CT_DisAction_2[1](xCycleStartMark:=Cy_lifter.xHP_Valve ,xCycleEndMark:= Cy_lifter.xHP_Delay,xCycleRun:=TRUE, RCycleTime=>ct_show.S01_CY_Lifter_HP);
CT_DisAction_2[2](xCycleStartMark:=Cy_lifter.xWP_Valve ,xCycleEndMark:= Cy_lifter.xWP_Delay,xCycleRun:=TRUE, RCycleTime=>ct_show.S01_CY_Lifter_WP);
CT_DisAction_2[3](xCycleStartMark:=Cy_rotate.xHP_Valve ,xCycleEndMark:= Cy_rotate.xHP_Delay,xCycleRun:=TRUE, RCycleTime=>ct_show.S01_CY_Rotate_HP);
CT_DisAction_2[4](xCycleStartMark:=Cy_rotate.xWP_Valve ,xCycleEndMark:= Cy_rotate.xWP_Delay,xCycleRun:=TRUE, RCycleTime=>ct_show.S01_CY_Rotate_WP);
CT_DisAction_2[5](xCycleStartMark:=Cy_takeClamp1.xHP_Valve ,xCycleEndMark:= Cy_takeClamp1.xHP_Delay,xCycleRun:=TRUE, RCycleTime=>ct_show.S01_Cy_takeClamp12_HP);
CT_DisAction_2[6](xCycleStartMark:=Cy_takeClamp1.xWP_Valve ,xCycleEndMark:= Cy_takeClamp1.xWP_Delay,xCycleRun:=TRUE, RCycleTime=>ct_show.S01_Cy_takeClamp12_WP);
CT_DisAction_2[7](xCycleStartMark:=Cy_takeClamp3.xHP_Valve ,xCycleEndMark:= Cy_takeClamp3.xHP_Delay,xCycleRun:=TRUE, RCycleTime=>ct_show.S01_Cy_takeClamp34_HP);
CT_DisAction_2[8](xCycleStartMark:=Cy_takeClamp3.xWP_Valve ,xCycleEndMark:= Cy_takeClamp3.xWP_Delay,xCycleRun:=TRUE, RCycleTime=>ct_show.S01_Cy_takeClamp34_WP);



//---------------------------------CV运行---------------------------------
 IF Machine_IO.xAutoMode THEN //自动模式下
	 IF station.xRunning THEN
		  Motion_ADD_cv_run[1]:=TRUE;//传送带运行置位
      Motion_ADD_cv_run[2]:=TRUE;   
   END_IF
END_IF
ft_cv(CLK:=station.xRunning AND  Machine_IO.xAutoMode , Q=> );
IF ft_cv.Q THEN
	 Motion_ADD_cv_run[1]:=FALSE;//传送带运行复位
   Motion_ADD_cv_run[2]:=FALSE;  
 END_IF
 
 //--------------------------------数据处理------------------------------
  rt_Clamp1HP(CLK:=Cy_takeClamp1.xHP_Delay, Q=> );
  rt_Clamp2HP(CLK:=Cy_takeClamp3.xHP_Delay , Q=> );
 //IF (rt_Clamp1HP.Q AND  Cy_rotate.xWP_Sensor) OR (rt_Clamp2HP.Q AND Cy_rotate.xHP_Sensor) THEN 	     
 IF station.xRunning AND NOT S05_CircleLine.Axis_Cycleline.xbusy THEN
   IF	 Sensor_Cycleline_on[1] OR (fbmachine[1].xTryRun) THEN
		 CardState[1].A:=TRUE;
		 CardState[1].Card_OK:=TRUE;	
   END_IF
   IF	 Sensor_Cycleline_on[2] OR (fbmachine[1].xTryRun) THEN
	 	 CardState[1].B:=TRUE;
		 CardState[1].Card_OK:=TRUE;	
	 END_IF
END_IF
END_ACTION

ACTION ILC:

//---------------------------------------------------工站可执行-------------------------------------------------------
station.xCanRun := TRUE ;

//---------------------------------------------------气缸动作条件-------------------------------------------
Cy_rotate.xOnILC:=Cy_lifter.xHP_Sensor OR Cy_rotate.xWP_Valve;
Cy_rotate.xOffILC:=Cy_lifter.xHP_Sensor OR Cy_rotate.xHP_Valve;

Cy_takeClamp1.xOnILC:=
Cy_takeClamp1.xOffILC:=TRUE;
                       //Cy_lifter.xWP_Delay 

//Cy_takeClamp2.xOnILC:=
//Cy_takeClamp2.xOffILC:=TRUE;

Cy_takeClamp3.xOnILC:=
Cy_takeClamp3.xOffILC:=TRUE;


//Cy_takeClamp4.xOnILC:=
//Cy_takeClamp4.xOffILC:=TRUE;

Cy_lifter.xOnILC:=NOT S05_CircleLine.Axis_Cycleline.xbusy AND Cy_rotate_on;
Cy_lifter.xOffILC:= TRUE ;
END_ACTION

ACTION TipAuto:

//------------------------------------------------AutoTip General---------------------------------


//------------------------------------------------AutoTip Cylinder--------------------------------

station.adwAutoTip[1].00:=FALSE;	//
station.adwAutoTip[1].01:=FALSE;	//
station.adwAutoTip[1].02:=Cy_rotate.xAutoTip;	       //Cy_rotate 气缸自动中有手动
station.adwAutoTip[1].03:=Cy_takeClamp1.xAutoTip;	   //Cy_takeClamp1 气缸自动中有手动
//station.adwAutoTip[1].04:=Cy_takeClamp2.xAutoTip;	   //Cy_takeClamp2 气缸自动中有手动
station.adwAutoTip[1].05:=Cy_takeClamp3.xAutoTip;	   //Cy_takeClamp3 气缸自动中有手动
//station.adwAutoTip[1].06:=Cy_takeClamp4.xAutoTip;	   //Cy_takeClamp4 气缸自动中有手动
station.adwAutoTip[1].07:=Cy_lifter	.xAutoTip;	     //Cy_lifter 气缸自动中有手动
END_ACTION

ACTION TipManual:
//--------------------------------------------ManualTip------------------------------------------------------
station.adwManualTip[1].00			:=FALSE;//提示1
//-------------------------------------------气缸提示---------------------------------------------------------




/////////////////////////////////////////////////////////////////////////////////////////////////////////////////
END_ACTION

END_PROGRAM

// Device/Application/POUS/02_STATION/S05_CircleLine
PROGRAM S05_CircleLine
VAR_INPUT

		//工站
	station					    : REFERENCE TO FB_Station:=fbStation[5];//工站状态
	cycleTime						: REFERENCE TO FB_CycleTime:= fbStCycleTime[5];	//工站CT
	//伺服
	Axis_Cycleline	    : REFERENCE TO FB_Axis:=fbAxis[1];
END_VAR
VAR
			arTon                 :ARRAY[1..10] OF ton ; 
			arTon_alarm           :ARRAY[1..10] OF ton ; 
		  cycle_data_switch     :R_TRIG;//数据切换信号
		  rt_Ctmark             :R_TRIG;
			i                     :INT;
			Transplant_Can        :BOOL;
			Bowlfeeder_Can        :BOOL;
			Pushcard_Can          :BOOL;
			Takebag_Can           :BOOL;
			Openbag_Can           :BOOL;			
			CT_DisAction          : ARRAY[1..10] OF FB_CycleTime;
			CT_DisAction_1        : ARRAY[1..10] OF FB_CycleTime_1;			
	  	CT_DisAction_2        : ARRAY[1..10] OF FB_CycleTime_2;			
END_VAR

Alarm();
Delay();
FlowAuto();
FlowInit();
General();
ILC();
TipAuto();
TipManual();

ACTION Alarm:
station.adwAlarm[1].00:=station.xInitTimeout;	             //工站初始化超时报警
station.adwAlarm[1].19:=	Axis_Cycleline.xError ;            //轴报错
station.adwAlarm[1].20:=	Axis_Cycleline.xNotPowerOn;         //未使能
station.adwAlarm[1].21:=	Axis_Cycleline.xMoveTimeout;        //定位超时
END_ACTION

ACTION Delay:

//----------------------------------------------动作延时-----------------------------------------------

arTon[1](IN:=  , PT:=T#10S , Q=> , ET=> );//排空计时
arTon[2](IN:=NOT CardState[1].Card_OK AND NOT Axis_Cycleline.xbusy AND xCycle_card_on , PT:=T#10S , Q=> , ET=> );//
arTon[3](IN:=   , PT:=T#60S , Q=> , ET=> );//
//----------------------------------------------报警延时-----------------------------------------------
arTon_alarm[1](IN:=NOT Axis_Cycleline.xbusy  , PT:=T#1S , Q=> , ET=> );//
arTon_alarm[2](IN:= , PT:=T#7S , Q=> , ET=> );//
arTon_alarm[3](IN:= , PT:=T#7S , Q=> , ET=> );//
arTon_alarm[4](IN:= , PT:=T#7S , Q=> , ET=> );//
arTon_alarm[5](IN:=   , PT:=T#60S , Q=> , ET=> );//
arTon_alarm[6](IN:=   , PT:=T#60S , Q=> , ET=> );//

arTon_alarm[7](IN:=   , PT:=T#10S , Q=> , ET=> );//
arTon_alarm[8](IN:=   , PT:=T#60S , Q=> , ET=> );//
arTon_alarm[9](IN:=   , PT:=T#60S , Q=> , ET=> );//
END_ACTION

ACTION FlowAuto:

//-----------------------------------------初始化是否完成判断----------------------------------------------
IF NOT station.xInitDone 
THEN
 	station.iStepAuto:=0;
 	station.xDone:=FALSE;
ELSIF station.xRunning  
THEN
//-----------------------------------------动作步骤--------------------------------------------------------
CASE station.iStepAuto OF	  
	0: //----Home Step，等待启动----
		
		IF station.xDisabled AND station.xCanRun 	AND NOT fbMachine[1].xStopped AND NOT station.xSingleRunning 
		THEN
			station.xDone:=TRUE;//工站完成信号判断
		END_IF
		
	  IF  station.xSingleRunning OR station.xCanRun	AND NOT station.xDone AND NOT station.xDisabled	AND NOT fbMachine[1].xStopped
		THEN
			station.xCycleEnable:=TRUE;
			station.xDone:= FALSE;  
			station.iStepAuto:= 60;
		END_IF

		40://启动前判断运行条件
		IF Axis_Cycleline.xRunILC AND S03_takebag.Axis_Cycleline.xRunILC THEN
	 //  S05_CycleLineMoveCount:= S05_CycleLineMoveCount +1;
	  	station.iStepAuto:= 50;
		END_IF	 
		50://启动
(*		 stData.Axis[1].rMovePosition[2] := stData.Axis[1].rMovePosition[1] +S05_CycleLineMoveCount* gc_rCycleLineSpacing;//200为两个节距
	   Axis_Cycleline.xMoveAuto[2]:=TRUE;//供袋环形线移动
    IF  Axis_Cycleline.xMoveInPos[2] THEN
				station.iStepAuto:= 999;  
		END_IF		
*)
    60:
		IF (Transplant_Can OR S01_transplant.station.xDisabled)
      AND (Bowlfeeder_Can OR S02_bowlFeeder.station.xDisabled) 
      AND (Pushcard_Can OR S04_PushCard.station.xDisabled)
      AND (Takebag_Can OR S03_takebag.station.xDisabled)
      AND (Openbag_Can OR  S06_OpenBag.station.xDisabled) AND NOT Axis_Cycleline.xbusy THEN		
		
		  station.iStepAuto :=70;
		END_IF

	70://数据处理
	IF NOT Axis_Cycleline.xbusy THEN
		Axis_Cycleline.xRelativeAuto:=TRUE;	
	END_IF
	IF Axis_Cycleline.xbusy THEN
		  FOR K :=8 TO 1 BY -1 DO
			CardState[K+1] := CardState[K] ;	
		  END_FOR  
			CardState[1]:=CardState[5]:=CardState[6];	//word 5 数据复位	
			station.iStepAuto :=80;
	END_IF
	80:	//等待完成	 
	  IF  Axis_Cycleline.xRelativeDone1  THEN
	    station.iStepAuto :=999;
		END_IF
	  999://----Single Run Finish----
		station.iStepAuto :=0;
		//station.xDone:=TRUE;
		station.xSingleRunFlag:=FALSE;
		station.xCycleEnable:=FALSE;	
END_CASE

END_IF
END_ACTION

ACTION FlowInit:
IF NOT station.xIniting THEN
  station.iStepInit:=0;    
ELSE
//--------------------------------------------初始化步序----------------------------------
CASE station.iStepInit OF	
 0://  
  	IF station.xIniting THEN	
  	  station.iStepInit:=10;	
  	END_IF	
10://复位数据
			CardState:= zero_card ;
      station.iStepInit := 20 ;		

20://轴上使能
   	Axis_Cycleline.xPowerInit := TRUE ;
    IF 	Axis_Cycleline.xPowerOn THEN 
    		station.iStepInit:=50;	
		END_IF		
50://轴回原点
    Axis_Cycleline.xHomeAuto := TRUE ;
		IF Axis_Cycleline.xHomeDone THEN
    Axis_Cycleline.xHomeAuto := FALSE ;
    		station.iStepInit:=60;	
		END_IF
60://轴去待机位
    Axis_Cycleline.xMoveAuto[1] := TRUE ;
		IF Axis_Cycleline.xMoveInPos[1] THEN 
    		station.iStepInit:=999;	
		END_IF			
999://初始化完成	
	station.iStepInit:=0;
	station.xInitDone:=TRUE;  
END_CASE
END_IF
END_ACTION

ACTION General:
//工站信息处理

(*IF station.xRunning THEN 
	//word 1有料判断，和传送复位
//传送时，数据交替	 
	 cycle_data_switch(CLK:=Axis_Cycleline.xMoveAuto[2], Q=> );
	 IF cycle_data_switch.Q THEN
		 FOR K :=8 TO 1 BY -1 DO
			CardState[K+1] := CardState[K] ;	
		  END_FOR  
		CardState[5]:=CardState[6];	//word 5 数据复位
	 END_IF 
END_IF
*)
//主轴停止状态
Axis_main_ready:=NOT Axis_Cycleline.xbusy;
//主轴上有料判断
IF CardState[1].Card_OK OR CardState[2].Card_OK OR CardState[3].Card_OK OR CardState[4].Card_OK  THEN
	xCycle_card_on:=TRUE;
	ELSE
	xCycle_card_on:=FALSE;	
END_IF
//周边工站完成信号复位
cycle_data_switch(CLK:=Axis_Cycleline.xbusy, Q=> );
IF cycle_data_switch.Q  THEN
	S01_transplant.station.xDone:=FALSE;
	S02_bowlFeeder.station.xDone:=FALSE;
//  S03_takebag.station.xDone:=FALSE;
	S04_PushCard.station.xDone:=FALSE;
//	S06_OpenBag.station.xDone:=FALSE;
END_IF
//自动排空处理
 //xCard_Empty:=TRUE;
 //点动数据，前进一节手动操作
 stData.Axis[1].rRelativeDistance:=gc_rCycleLineSpacing;
 
//CT
rt_Ctmark(CLK:=Axis_Cycleline.xRelativeAuto, Q=>cycleTime.xCycleMark );   
 
CT_DisAction[1](xCycleMark:=Axis_Cycleline.xbusy,xCycleRun:=TRUE,rCycleTime=>);
CT_DisAction[2](xCycleMark:=NOT Bowlfeeder_Can,xCycleRun:=TRUE,rCycleTime=>);
CT_DisAction[3](xCycleMark:=NOT Takebag_Can,xCycleRun:=TRUE,rCycleTime=>);
CT_DisAction[4](xCycleMark:=NOT Pushcard_Can,xCycleRun:=TRUE,rCycleTime=>);
CT_DisAction[5](xCycleMark:=NOT Openbag_Can,xCycleRun:=TRUE,rCycleTime=>);
CT_DisAction[6](xCycleMark:=Axis_Cycleline.xRelativeAuto,xCycleRun:=TRUE, RCycleTime=>ct_show.S05_Total);

CT_DisAction_1[1](xCycleMark:=Axis_Cycleline.xbusy,xCycleRun:=TRUE, RCycleTime=>ct_show.S05_AXIS_Relative);

//工站运行条件可
//S01
IF (CardState[1].Card_OK OR arTon[2].Q OR S01_transplant.station.xDisabled ) AND  S01_transplant.Cy_lifter.xHP_Delay  THEN
	Transplant_Can:=TRUE;
	ELSE
	Transplant_Can:=FALSE;
END_IF
//S02
IF CardState[2].Desiccant_OK OR NOT CardState[2].Card_OK OR S02_bowlFeeder.station.xDisabled THEN
	Bowlfeeder_Can:=TRUE;
	ELSE
	Bowlfeeder_Can:=FALSE;
END_IF
//S03
IF (BagState[1].Takebag_OK OR NOT CardState[2].Card_OK OR S03_takebag.station.xDisabled) AND S03_takebag.Cy_lifter.xHP_Delay  THEN
	Takebag_Can:=TRUE;
	ELSE
	Takebag_Can:=FALSE;
END_IF
//S04
IF (CardState[4].Pushcard_OK OR NOT CardState[4].Card_OK OR S04_PushCard.station.xDisabled) AND S04_PushCard.Cy_push1.xHP_Delay AND S04_PushCard.Cy_push2.xHP_Delay  THEN
	Pushcard_Can:=TRUE;
	ELSE
	Pushcard_Can:=FALSE;
END_IF
//S06
IF BagState[2].Suck_OK OR NOT CardState[3].Card_OK OR S06_OpenBag.station.xDisabled   THEN
	Openbag_Can:=TRUE;
	ELSE
	Openbag_Can:=FALSE;
END_IF
END_ACTION

ACTION ILC:

//---------------------------------------------------工站可执行-------------------------------------------------------
station.xCanRun := TRUE ;

//---------------------------------------------------气缸动作条件-------------------------------------------



//---------------------------------------------------伺服动作条件-------------------------------------------
	Axis_Cycleline.xJogILC := TRUE;    
	Axis_Cycleline.xHomeILC := 
	Axis_Cycleline.xRunILC := 
	Axis_Cycleline.xRelativeILC:=
	Axis_Cycleline.xMoveILC[1] :=                           
	Axis_Cycleline.xMoveILC[2] :=                           
	Axis_Cycleline.xMoveILC[3] :=  S01_transplant.Cy_lifter.xHP_Sensor //S01移栽气缸原点
                          AND (NOT S02_bowlFeeder.Axis_PPU.xMoveInPos[2] AND NOT S02_bowlFeeder.Axis_PPU.xbusy) //S02模组保护
                          AND  S06_OpenBag.Cy_lifter_HPSensor AND S04_PushCard.Cy_push1.xHP_Sensor AND S04_PushCard.Cy_push2.xHP_Sensor;//S04推料和盖板气缸原点
   //联动保护在自动流程里面
END_ACTION

ACTION TipAuto:

//------------------------------------------------AutoTip General---------------------------------


//------------------------------------------------AutoTip Cylinder--------------------------------

station.adwAutoTip[1].00:=FALSE;	//
station.adwAutoTip[1].01:=FALSE;	//
//伺服位置的读取,伺服位置错误自动提示               //Axis_distributor自动时位置错误
   FOR i:= 1 TO 5 BY 1 DO 
   	IF Axis_Cycleline.xMoveAuto[i] THEN
   		Axis_Cycleline.iPosNumber := i ;
   	END_IF
   END_FOR
(*IF fbMachine[1].xAutoMode AND NOT fbMachine[1].xRunning AND arTon_alarm[1].Q THEN 
	IF Axis_Cycleline.iPosNumber=1 AND NOT Axis_Cycleline.xMoveInPos[1] THEN station.adwAutoTip[1].08:=TRUE; END_IF //轴自动时位置不在位置1
	IF Axis_Cycleline.iPosNumber=2 AND NOT Axis_Cycleline.xMoveInPos[2] THEN station.adwAutoTip[1].09:=TRUE; END_IF //轴自动时位置不在位置2
	IF Axis_Cycleline.iPosNumber=3 AND NOT Axis_Cycleline.xMoveInPos[3] THEN station.adwAutoTip[1].10:=TRUE; END_IF //轴自动时位置不在位置3
END_IF
*)
END_ACTION

ACTION TipManual:
//--------------------------------------------ManualTip------------------------------------------------------
station.adwManualTip[1].00			:=FALSE;//提示1
//-------------------------------------------气缸提示---------------------------------------------------------




/////////////////////////////////////////////////////////////////////////////////////////////////////////////////
END_ACTION

END_PROGRAM

// Device/Application/POUS/02_STATION/S03_takebag
PROGRAM S03_takebag
VAR_INPUT
	//工站
	station					    : REFERENCE TO FB_Station:=fbStation[3];//工站状态
	cycleTime						: REFERENCE TO FB_CycleTime:= fbStCycleTime[3];	//工站CT
  //伺服
	Axis_Cycleline	  : REFERENCE TO FB_Axis:=fbAxis[2];

 //气缸
	 Cy_lifter				      : REFERENCE TO FB_Cylinder:=fbCylinder[11];//取袋-升降
	//真空发生器
		Va_take1				      : REFERENCE TO FB_Vacuum:=fbVacuum[3];     //取袋真空1
		Va_take2				      : REFERENCE TO FB_Vacuum:=fbVacuum[4];     //取袋真空2	
	//传感器
	Sensor_lackbag            : ARRAY[1..2] OF BOOL; //缺袋检测
	Sensor_BagOn              : ARRAY[1..2] OF BOOL; //有袋检测
END_VAR
//内部变量
VAR
			arTon               :ARRAY[1..10] OF ton ;
      arTon_alarm         :ARRAY[1..10] OF ton ;  
			iOpen_bag_Step      :INT;
			rg_cycle_run        :R_TRIG;
      rt_Ctmark           :R_TRIG;
			i                   :INT;
			CT_DisAction          : ARRAY[1..10] OF FB_CycleTime;
			CT_DisAction_1        : ARRAY[1..10] OF FB_CycleTime_1;			
	  	CT_DisAction_2        : ARRAY[1..10] OF FB_CycleTime_2;		
END_VAR

Alarm();
Delay();
FlowAuto();
FlowInit();
General();
ILC();
TipAuto();
TipManual();

ACTION Alarm:
//ALARM
station.adwAlarm[1].00:=station.xInitTimeout;	             //Add_distributor 工站初始化超时报警
station.adwAlarm[1].01:=	Cy_lifter.xHP_Off ;        //Add_distributor Cy_takeClamp1_1 气缸原点无信号
station.adwAlarm[1].02:=	Cy_lifter.xWP_Off ;        //Add_distributor Cy_takeClamp1_1 气缸动点无信号
station.adwAlarm[1].03:=	Va_take1.byAlarm.1;         //吸真空报警
station.adwAlarm[1].04:=	Va_take1.byAlarm.3 ;        //破真空报警
station.adwAlarm[1].05:=	Va_take2.byAlarm.1 ;        //
station.adwAlarm[1].06:=	Va_take2.byAlarm.3 ;   
station.adwAlarm[1].07:=	Axis_Cycleline.xError ;            //轴报错
station.adwAlarm[1].08:=	Axis_Cycleline.xNotPowerOn;         //未使能
station.adwAlarm[1].09:=	Axis_Cycleline.xMoveTimeout;        //定位超时


//WARNING
IF NOT fbmachine[1].xTryRun THEN
station.adwWarning[1].00:=arTon_alarm[1].Q;//缺袋1
station.adwWarning[1].01:=arTon_alarm[2].Q;//缺袋2
END_IF
END_ACTION

ACTION Delay:

//----------------------------------------------动作延时-----------------------------------------------

arTon[1](IN:=((Va_take1.xVacuumSensor OR NOT CardState[2].A) AND  (Va_take2.xVacuumSensor OR NOT CardState[2].B)  OR fbmachine[1].xTryRun) AND station.iStepAuto=15, PT:=T#100MS , Q=> , ET=> );//防止真空信号有时差
arTon[2](IN:=  , PT:=T#3S , Q=> , ET=> );//
arTon[3](IN:=  , PT:=T#1S , Q=> , ET=> );//
arTon[4](IN:=   , PT:=T#60S , Q=> , ET=> );//
arTon[5](IN:=   , PT:=T#60S , Q=> , ET=> );//
arTon[6](IN:=   , PT:=T#60S , Q=> , ET=> );//
//----------------------------------------------报警延时-----------------------------------------------
arTon_alarm[1](IN:= station.xRunning AND NOT Sensor_lackbag[1] , PT:=T#1S , Q=> , ET=> );//缺袋检测1
arTon_alarm[2](IN:= station.xRunning AND NOT Sensor_lackbag[2] , PT:=T#1S , Q=> , ET=> );//缺袋检测2
arTon_alarm[3](IN:=NOT Axis_Cycleline.xbusy , PT:=T#1S , Q=> , ET=> );//
arTon_alarm[4](IN:= , PT:=T#7S , Q=> , ET=> );//
arTon_alarm[5](IN:=   , PT:=T#60S , Q=> , ET=> );//
arTon_alarm[6](IN:=   , PT:=T#60S , Q=> , ET=> );//

arTon_alarm[7](IN:=   , PT:=T#10S , Q=> , ET=> );//
arTon_alarm[8](IN:=   , PT:=T#60S , Q=> , ET=> );//
arTon_alarm[9](IN:=   , PT:=T#60S , Q=> , ET=> );//
END_ACTION

ACTION FlowAuto:

//-----------------------------------------初始化是否完成判断----------------------------------------------
IF NOT station.xInitDone 
THEN
 	station.iStepAuto:=0;
 	station.xDone:=FALSE;
ELSIF station.xRunning  // OR station.xSingleRunFlag //HMI触发单循环
THEN
//-----------------------------------------动作步骤--------------------------------------------------------
CASE station.iStepAuto OF	  
	0: //----Home Step，等待启动----
		
		IF station.xDisabled AND station.xCanRun 	AND NOT fbMachine[1].xStopped AND NOT station.xSingleRunning 
		THEN
			station.xDone:=TRUE;//工站完成信号判断
		END_IF
		
	  IF  station.xSingleRunning OR station.xCanRun	AND NOT station.xDone AND NOT station.xDisabled	AND NOT fbMachine[1].xStopped
		THEN
			station.xCycleEnable:=TRUE;
			station.xDone:= FALSE;  
			station.iStepAuto:= 5;
		END_IF
		5://数据复位			
		  station.iStepAuto:= 10;
//取袋流程
	 	10://判断顶升
		IF NOT Axis_Cycleline.xbusy AND (NOT BagState[1].Takebag_OK OR station.xSingleRunFlag) AND (CardState[2].Card_OK OR fbmachine[1].xTryRun OR station.xSingleRunFlag)
      THEN
			Cy_lifter.xAuto:=TRUE;		
		END_IF
		IF Cy_lifter.xWP_Delay THEN
	  	  station.iStepAuto:= 15;		
	 	END_IF			
    IF 	BagState[1].Takebag_OK THEN
        station.iStepAuto:= 40;		
		END_IF
	   15://判断取袋
		  IF NOT fbmachine[1].xTryRun THEN
		    IF CardState[2].A OR station.xSingleRunFlag THEN
						Va_take1.xVacuumAuto:=TRUE;	
		  	END_IF
		    IF CardState[2].B OR station.xSingleRunFlag THEN
						Va_take2.xVacuumAuto:=TRUE;	
		  	END_IF	 
			END_IF
		  IF arTon[1].Q THEN//可以全部不取，取决于主环形线
			  station.iStepAuto:= 20;				 
  	   END_IF   	 	 
		 20://放到传送带
	   	Cy_lifter.xAuto:=FALSE;	
			IF Cy_lifter.xHP_Delay AND (Sensor_BagOn[1] OR Sensor_BagOn[2] OR fbmachine[1].xTryRun) THEN
	    	Va_take1.xVacuumAuto:=FALSE;	
		   	Va_take2.xVacuumAuto:=FALSE;
		  	 station.iStepAuto:= 30;	
			END_IF
    30://取袋完成
			IF  NOT (Va_take1.xVacuumDelay OR  Va_take2.xVacuumDelay)  THEN
			 BagState[1].Takebag_OK:=TRUE;
			 station.iStepAuto:= 40;	
			END_IF
		40://环线线动作
      IF  NOT  Axis_Cycleline.xbusy AND ((BagState[2].Suck_OK OR NOT BagState[2].Takebag_OK)  AND  S05_CircleLine.Axis_Cycleline.xbusy) OR station.xSingleRunFlag THEN
		       Axis_Cycleline.xRelativeAuto:=TRUE;
					 station.iStepAuto:= 50;
		  END_IF
	  50://数据传递
		IF Axis_Cycleline.xbusy THEN
		  FOR K :=8 TO 1 BY -1 DO
			 BagState[K+1] := BagState[K] ;		 
		  END_FOR
		  BagState[1]:=BagState[4]:=BagState[5];	//工站4 数据复位
      station.iStepAuto:= 60;	
	  END_IF
		60:// 
		 IF  Axis_Cycleline.xRelativeDone1   //Axis_Cycleline.xMoveInPos[2]
     THEN
				 station.iStepAuto:= 999;	
     END_IF
		
		
		
	999://----Single Run Finish----
			
		station.iStepAuto :=0;
	//	station.xDone:=TRUE;
		station.xSingleRunFlag:=FALSE;
		station.xCycleEnable:=FALSE;	
END_CASE

END_IF
END_ACTION

ACTION FlowInit:
IF NOT station.xIniting THEN
  station.iStepInit:=0;    
ELSE
//--------------------------------------------初始化步序----------------------------------
CASE station.iStepInit OF	
 0://  
  	IF station.xIniting THEN	
  	  station.iStepInit:=10;	
  	END_IF	
10://复位数据
    BagState[1].Takebag_OK:=TRUE;
		BagState:= zero_bag ;
    station.iStepInit := 20 ;		
20://真空复位
      Va_take1.xVacuumAuto := 
      Va_take1.xBreakAuto := 
			Va_take1.xVacuumManual:=FALSE;
      Va_take2.xVacuumAuto := 
      Va_take2.xBreakAuto := 
			Va_take2.xVacuumManual:=FALSE;
			station.iStepInit:=30;	
 30://
    Cy_lifter.xInit := TRUE ;
		IF Cy_lifter.xHP_Delay   THEN 
    station.iStepInit:=40;	
		END_IF		
 40://轴上使能
    	Axis_Cycleline.xPowerInit := TRUE ;
		
    IF 	Axis_Cycleline.xPowerOn  THEN 
    		station.iStepInit:=50;	
		END_IF		
50://轴回原点-绝对值
    Axis_Cycleline.xHomeAuto := TRUE ;

		IF Axis_Cycleline.xHomeDone  THEN
       Axis_Cycleline.xHomeAuto := FALSE ;
		
    		station.iStepInit:=60;	
		END_IF
60://轴去待机位
    Axis_Cycleline.xMoveAuto[1] := TRUE ;
	 
		IF Axis_Cycleline.xMoveInPos[1] THEN 
    		station.iStepInit:=999;	
		END_IF	
 
 

			
999://初始化完成	
	station.iStepInit:=0;
	station.xInitDone:=TRUE;  
END_CASE
END_IF
END_ACTION

ACTION General:


 //点动数据
stData.Axis[2].rRelativeDistance:=gc_rCycleLineSpacing;

//CT
rt_Ctmark(CLK:=Cy_lifter.xAuto , Q=>cycleTime.xCycleMark );


CT_DisAction_2[1](xCycleStartMark:=Cy_lifter.xHP_Valve ,xCycleEndMark:= Cy_lifter.xHP_Delay,xCycleRun:=TRUE, RCycleTime=>ct_show.s03_CY_Lifter_HP);
CT_DisAction_2[2](xCycleStartMark:=Cy_lifter.xWP_Valve ,xCycleEndMark:= Cy_lifter.xWP_Delay,xCycleRun:=TRUE, RCycleTime=>ct_show.s03_CY_Lifter_WP);
CT_DisAction_2[3](xCycleStartMark:=Axis_Cycleline.xRelativeAuto ,xCycleEndMark:= Axis_Cycleline.xRelativeDone1,xCycleRun:=TRUE, RCycleTime=>ct_show.S03_AXIS_Relative);
END_ACTION

ACTION ILC:

//---------------------------------------------------工站可执行-------------------------------------------------------
station.xCanRun := TRUE ;

//---------------------------------------------------气缸动作条件-------------------------------------------


Cy_lifter.xOnILC:=
Cy_lifter.xOffILC:=TRUE;






//---------------------------------------------------伺服动作条件-------------------------------------------
	Axis_Cycleline.xJogILC := TRUE;    
	Axis_Cycleline.xHomeILC := 
	Axis_Cycleline.xRunILC := 
	Axis_Cycleline.xRelativeILC:=
	Axis_Cycleline.xMoveILC[1] :=                         //取料位
	Axis_Cycleline.xMoveILC[2] :=
	Axis_Cycleline.xMoveILC[3] :=Cy_lifter.xHP_Sensor;
END_ACTION

ACTION TipAuto:

//------------------------------------------------AutoTip General---------------------------------


//------------------------------------------------AutoTip Cylinder--------------------------------

station.adwAutoTip[1].00:=FALSE;	//
station.adwAutoTip[1].01:=FALSE;	//
station.adwAutoTip[1].02:=Cy_lifter.xAutoTip;	   //升降气缸自动中有手动
station.adwAutoTip[1].03:=FALSE;	   //取料真空1自动中有手动
station.adwAutoTip[1].04:=FALSE;	   //取料真空2自动中有手动

//伺服位置的读取,伺服位置错误自动提示               //Axis_distributor自动时位置错误
   FOR i:= 1 TO 5 BY 1 DO 
   	IF Axis_Cycleline.xMoveAuto[i] THEN
   		Axis_Cycleline.iPosNumber := i ;
   	END_IF
   END_FOR
(*IF fbMachine[1].xAutoMode AND NOT fbMachine[1].xRunning AND arTon_alarm[3].Q THEN 
	IF Axis_Cycleline.iPosNumber=1 AND NOT Axis_Cycleline.xMoveInPos[1] THEN station.adwAutoTip[1].05:=TRUE; END_IF //轴自动时位置不在位置1
	IF Axis_Cycleline.iPosNumber=2 AND NOT Axis_Cycleline.xMoveInPos[2] THEN station.adwAutoTip[1].06:=TRUE; END_IF //轴自动时位置不在位置2
	IF Axis_Cycleline.iPosNumber=3 AND NOT Axis_Cycleline.xMoveInPos[3] THEN station.adwAutoTip[1].07:=TRUE; END_IF //轴自动时位置不在位置3
END_IF*)
END_ACTION

ACTION TipManual:
//--------------------------------------------ManualTip------------------------------------------------------
station.adwManualTip[1].00			:=FALSE;//提示1
//-------------------------------------------气缸提示---------------------------------------------------------




/////////////////////////////////////////////////////////////////////////////////////////////////////////////////
END_ACTION

END_PROGRAM

// Device/Application/FB/16_VacuumFB/FB_Vacuum
FUNCTION_BLOCK FB_Vacuum
VAR_INPUT
	xManualMode					: BOOL;					//手动模式
	xAirOn						: BOOL;					//气压正常
	xReset						: BOOL;					//复位
	xAlarmDisable               : BOOL ;                //真空报警屏蔽
	xVacuumHmi					: BOOL;					//吸真空HMI
	xVacuumManual				: BOOL;					//吸真空手动执行
	xVacuumAuto					: BOOL;					//吸真空自动执行
	xBreakHmi					: BOOL;					//破真空HMI
	xBreakManual				: BOOL;					//破真空手动执行
	xBreakAuto					: BOOL;					//破真空自动执行
	xVacuumSensor				: BOOL;					//真空感应器
	tAlarm						: TIME:=T#5S;			//报警延时			//取料真空报警优化
	tBreakDelay					: (*REFERENCE TO*) TIME;	//破真空延时
	tVacuumDelay				: (*REFERENCE TO*) TIME;//;	//吸真空延时
END_VAR

VAR_OUTPUT
	xVacuumValve				: BOOL;					//吸真空阀输出
	xBreakValve					: BOOL;					//破真空阀输出
	xVacuumDelay				: BOOL;					//吸真空状态
	xBreakDelay					: BOOL;					//破真空状态
	byAlarm						: BYTE;					 //报警字节,bit1:吸真空感应器无信号,3:吸真空感应器有信号
END_VAR

VAR
	{attribute 'hide'}
	ftBreakHmi					: F_TRIG;				//破真空HMI下降沿
	{attribute 'hide'}
	ftVacuumHmi					: F_TRIG;				//吸真空HMI下降沿
	{attribute 'hide'}
	tonBreakDelay				: TON;					//破真空延时计时
	{attribute 'hide'}
	tonVacuumDelay				: TON;					//吸真空延时计时
	{attribute 'hide'}
	tonAlarm					: TON;					//报警延时计时
END_VAR

ACT_Manual();
ACT_Output();
ACT_Delay();
ACT_Alarm();

ACTION ACT_Alarm:
//	报警延时
tonAlarm(
	IN:=xAirOn
	    AND NOT xReset
		AND NOT xAlarmDisable
		AND (xVacuumValve AND NOT xVacuumDelay
			OR xBreakValve AND NOT xBreakDelay
		),
	PT:=tAlarm + MAX(tBreakDelay, tVacuumDelay),
	Q=>, ET=>);

//	报警复位
IF xReset 
	OR xAlarmDisable 				//吸取失败处理
THEN
	byAlarm:=0;
END_IF

//--------------------------报警输出---------------
IF tonAlarm.Q 
	AND xAirOn
THEN
//吸真空异常
	IF xVacuumValve AND NOT xVacuumSensor THEN
		byAlarm.1:=TRUE;
	END_IF
//破真空异常	
	IF xBreakValve AND xVacuumSensor THEN
		byAlarm.3:=TRUE;
	END_IF
END_IF
END_ACTION

ACTION ACT_Delay:
//	破真空延时
tonBreakDelay(
	IN:=xAirOn
		AND xBreakValve
		AND NOT xVacuumValve
		AND NOT xVacuumSensor,
	PT:=tBreakDelay,
	Q=>xBreakDelay,
	ET=>);

//	吸真空延时
tonVacuumDelay(
	IN:=xAirOn
		AND NOT xBreakValve
		AND xVacuumValve
		AND xVacuumSensor,
	PT:=tVacuumDelay,
	Q=>xVacuumDelay,
	ET=>);
END_ACTION

ACTION ACT_Manual:
//	手动操作
ftVacuumHmi(CLK:=xVacuumHmi, Q=>);
ftBreakHmi(CLK:=xBreakHmi, Q=>);
IF xManualMode	AND xAirOn
THEN
	IF ftVacuumHmi.Q		AND NOT xBreakAuto
	THEN
		xVacuumManual:=NOT xVacuumManual;
		xBreakManual:=FALSE;
	END_IF
	IF ftBreakHmi.Q		AND NOT xVacuumAuto
	THEN
		xBreakManual:=NOT xBreakManual;
		xVacuumManual:=FALSE;
	END_IF
END_IF

IF NOT xManualMode THEN
	xBreakManual:=FALSE;
	xVacuumManual:=FALSE;
END_IF
END_ACTION

ACTION ACT_Output:
(*
//	吸真空阀输出
bVacuumValve:=NOT bBreakValve
	AND (bVacuumManual
		OR bVacuumAuto);

//	破真空阀输出
bBreakValve:=NOT bVacuumValve
	AND (bBreakManual
		OR bBreakAuto);
*)
//	破真空阀输出
xBreakValve:=NOT xVacuumValve AND (xBreakAuto AND NOT xManualMode)
							OR (xBreakManual XOR xBreakAuto AND xManualMode);

//	吸真空阀输出
xVacuumValve:=NOT xBreakValve AND ( xVacuumAuto AND NOT xManualMode)
							OR (xVacuumManual XOR xVacuumAuto AND xManualMode);
END_ACTION

END_FUNCTION_BLOCK

// Device/Application/POUS/02_STATION/S02_bowlFeeder
PROGRAM S02_bowlFeeder
VAR_INPUT
//工站
	station					    : REFERENCE TO FB_Station:=fbStation[2];//工站状态
	cycleTime						: REFERENCE TO FB_CycleTime:= fbStCycleTime[2];	//工站CT
//伺服
	Axis_PPU	          : REFERENCE TO FB_Axis:=fbAxis[4];
//气缸
	Cy_resist_1				    : REFERENCE TO FB_Cylinder:=fbCylinder[7];//阻挡气缸1-通道1
	Cy_resist_2				    : REFERENCE TO FB_Cylinder:=fbCylinder[8];//阻挡气缸2-通道1
	Cy_resist_3				    : REFERENCE TO FB_Cylinder:=fbCylinder[9];//阻挡气缸1-通道2
	Cy_resist_4				    : REFERENCE TO FB_Cylinder:=fbCylinder[10];//阻挡气缸2-通道2
//真空发生器
  Va_ppu_1				      : REFERENCE TO FB_Vacuum:=fbVacuum[1];     //PPU模组吸真空1
  Va_ppu_2				      : REFERENCE TO FB_Vacuum:=fbVacuum[2];     //PPU模组吸真空1	
//传感器
	Sensor_cv_on                   : ARRAY[1..2] OF BOOL; //传送带到位信号
	Sensor_Cycleline_on            : ARRAY[1..2] OF BOOL; //环形线放置到位
	Sensor_resist                  : ARRAY[1..4] OF BOOL; //干燥剂阻挡传感器
	Sensor_PPU_P                   : BOOL;//PPU正限位
  Sensor_PPU_H                   : BOOL;//PPU原点
	Sensor_PPU_N                   : BOOL;//PPU负限位

END_VAR
//内部变量
VAR
			arTon               :ARRAY[1..10] OF ton ; 
			arTon_alarm         :ARRAY[1..10] OF ton ; 
      rt_Ctmark           :R_TRIG;			
			i                   :INT;
			ft_cv               :F_TRIG;
			CESHI               :BOOL;
			resist_open         :ARRAY[1..4] OF BOOL;
			CT_DisAction          : ARRAY[1..10] OF FB_CycleTime;
			CT_DisAction_1        : ARRAY[1..10] OF FB_CycleTime_1;			
	  	CT_DisAction_2        : ARRAY[1..10] OF FB_CycleTime_2;
END_VAR

Alarm();
Delay();
FlowAuto();
FlowInit();
General();
ILC();
TipAuto();
TipManual();

ACTION TipManual:
//--------------------------------------------ManualTip------------------------------------------------------
station.adwManualTip[1].00			:=FALSE;//提示1
//-------------------------------------------气缸提示---------------------------------------------------------




/////////////////////////////////////////////////////////////////////////////////////////////////////////////////
END_ACTION

ACTION Alarm:
station.adwAlarm[1].00:=station.xInitTimeout;	             //Add_distributor 工站初始化超时报警
station.adwAlarm[1].01:=	Cy_resist_1.xHP_Off ;        //气缸原点无信号
station.adwAlarm[1].02:=	Cy_resist_1.xWP_Off ;        //气缸动点无信号
station.adwAlarm[1].03:=	Cy_resist_2.xHP_Off ;        //
station.adwAlarm[1].04:=	Cy_resist_2.xWP_Off ;        //
station.adwAlarm[1].05:=	Cy_resist_3.xHP_Off ;        //
station.adwAlarm[1].06:=	Cy_resist_3.xWP_Off ;        //
station.adwAlarm[1].07:=	Cy_resist_4.xHP_Off ;        //
station.adwAlarm[1].08:=	Cy_resist_4.xWP_Off;         //
station.adwAlarm[1].09:=	Va_ppu_1.byAlarm.1 ;         //吸真空报警
station.adwAlarm[1].10:=	Va_ppu_1.byAlarm.3 ;         //破真空报警
station.adwAlarm[1].11:=	Va_ppu_2.byAlarm.1 ;        //
station.adwAlarm[1].12:=	Va_ppu_2.byAlarm.3 ;        //
station.adwAlarm[1].13:=	Axis_PPU.xError ;            //轴报错
station.adwAlarm[1].14:=	Axis_PPU.xNotPowerOn;         //未使能
station.adwAlarm[1].15:=	Axis_PPU.xMoveTimeout;        //定位超时
END_ACTION

ACTION Delay:

//----------------------------------------------动作延时-----------------------------------------------

arTon[1](IN:= NOT Sensor_cv_on[1]  , PT:=T#1S , Q=> , ET=> );//控制阻挡气缸节拍		
arTon[2](IN:= NOT Sensor_cv_on[2]  , PT:=T#1S , Q=> , ET=> );//控制阻挡气缸节拍		 
arTon[3](IN:=((Va_ppu_1.xVacuumSensor OR NOT CardState[2].A) AND  (Va_ppu_2.xVacuumSensor OR NOT CardState[2].B) OR fbmachine[1].xTryRun )AND station.iStepAuto=15, PT:=T#300MS , Q=> , ET=> );//OR fbmachine[1].xTryRun 防止真空信号有时差
arTon[4](IN:= NOT resist_open[1]  , PT:=T#0.5S , Q=> , ET=> );//阻挡气缸1延时落下
arTon[5](IN:= NOT resist_open[2]  , PT:=T#0.5S , Q=> , ET=> );//阻挡气缸2延时落下
arTon[6](IN:= NOT resist_open[3]  , PT:=T#0.5S , Q=> , ET=> );//阻挡气缸3延时落下
arTon[7](IN:= NOT resist_open[4]  , PT:=T#0.5S , Q=> , ET=> );//阻挡气缸4延时落下
//----------------------------------------------报警延时-----------------------------------------------
arTon_alarm[1](IN:= NOT Axis_PPU.xbusy, PT:=T#1S , Q=> , ET=> );//轴到位判断延时
arTon_alarm[2](IN:= , PT:=T#7S , Q=> , ET=> );//
arTon_alarm[3](IN:= , PT:=T#7S , Q=> , ET=> );//
arTon_alarm[4](IN:= , PT:=T#7S , Q=> , ET=> );//
arTon_alarm[5](IN:=   , PT:=T#60S , Q=> , ET=> );//
arTon_alarm[6](IN:=   , PT:=T#60S , Q=> , ET=> );//

arTon_alarm[7](IN:=   , PT:=T#10S , Q=> , ET=> );//
arTon_alarm[8](IN:=   , PT:=T#60S , Q=> , ET=> );//
arTon_alarm[9](IN:=   , PT:=T#60S , Q=> , ET=> );//
END_ACTION

ACTION FlowAuto:

//-----------------------------------------初始化是否完成判断----------------------------------------------
IF NOT station.xInitDone 
THEN
 	station.iStepAuto:=0;
 	station.xDone:=FALSE;
ELSIF station.xRunning  
THEN
//-----------------------------------------动作步骤--------------------------------------------------------
CASE station.iStepAuto OF	  
	0: //----Home Step，等待启动----
		
		IF station.xDisabled AND station.xCanRun 	AND NOT fbMachine[1].xStopped AND NOT station.xSingleRunning 
		THEN
			station.xDone:=TRUE;//工站完成信号判断
		END_IF
		
	  IF  station.xSingleRunning OR station.xCanRun	AND NOT station.xDone AND NOT station.xDisabled	AND NOT fbMachine[1].xStopped
		THEN
			station.xCycleEnable:=TRUE;
			station.xDone:= FALSE;  
			station.iStepAuto:= 5;
		END_IF
		5://数据复位
				station.iStepAuto:= 10;
		10://PPU模组取料   根据实际取料去取料位------带料空跑修改点
		IF Axis_PPU.xMoveInPos[1] AND (CardState[2].Card_OK  AND NOT CardState[2].Desiccant_OK OR station.xSingleRunFlag) AND (sensor_cv_on[1] AND sensor_cv_on[2]OR  fbmachine[1].xTryRun)
      THEN 
     Axis_PPU.xMoveAuto[3]:=TRUE;
		END_IF
		IF Axis_PPU.xMoveInPos[3] THEN
			station.iStepAuto:= 15;
		END_IF

		15://取料
    IF NOT fbmachine[1].xTryRun  THEN//带料空跑修改点
	  	   IF (CardState[2].A OR station.xSingleRunFlag) AND sensor_cv_on[1] THEN
					  Va_ppu_1.xVacuumAuto:=TRUE;
				 END_IF
				 IF (CardState[2].B OR station.xSingleRunFlag) AND sensor_cv_on[2] THEN
		      	Va_ppu_2.xVacuumAuto:=TRUE;			
	       END_IF
  	 END_IF
		IF arTon[3].Q  AND NOT Axis_PPU.xbusy THEN
			station.iStepAuto:= 20;
		END_IF
		20://
		Axis_PPU.xMoveAuto[2]:=TRUE;
		IF Axis_PPU.xMoveInPos[2] THEN
			station.iStepAuto:= 25;
		END_IF
    25: //放料
		IF  NOT S05_CircleLine.Axis_Cycleline.xbusy AND Axis_PPU.xMoveInPos[2] THEN
			Va_ppu_1.xVacuumAuto:=FALSE;
			Va_ppu_2.xVacuumAuto:=FALSE;	
		END_IF
		IF NOT (Va_ppu_1.xVacuumSensor OR Va_ppu_2.xVacuumSensor ) THEN
			station.iStepAuto:= 30;
		END_IF
		
		30://数据处理
		IF   fbmachine[1].xTryRun OR Sensor_Cycleline_on[1] OR Sensor_Cycleline_on[2] OR Axis_PPU.xMoveInPos[2]
       THEN
			 CardState[2].Desiccant_OK:=TRUE;
			 station.iStepAuto:= 40;
		END_IF	
		40://回去取料位
		IF 	 NOT Axis_PPU.xbusy   THEN
			Axis_PPU.xMoveAuto[1]:=TRUE;
		END_IF
		IF Axis_PPU.xMoveInPos[1] THEN
						station.iStepAuto:= 999;
		END_IF
		
		
		
		
		
		
		
	999://----Single Run Finish----
			
		station.iStepAuto :=0;
  	station.xDone:=TRUE;
		station.xSingleRunFlag:=FALSE;
		station.xCycleEnable:=FALSE;	
END_CASE

END_IF
END_ACTION

ACTION FlowInit:
IF NOT station.xIniting THEN
  station.iStepInit:=0;    
ELSE
//--------------------------------------------初始化步序----------------------------------
CASE station.iStepInit OF	
 0://  
  	IF station.xIniting THEN	
			CardState[2].Desiccant_OK:=FALSE;
  	  station.iStepInit:=10;	
  	END_IF	
10://复位数据
    Motion_S02_cv_run:=FALSE;//传送带运行复位   
    Box_blow[1]:=FALSE;
    Box_blow[2]:=FALSE; 
    Box_run :=FALSE; 
    station.iStepInit := 20 ;		
20://升降气缸原点
 //  IF NOT Sensor_resist[1] THEN
		 Cy_resist_1.xInit:=TRUE;
	// END_IF  
//   IF NOT Sensor_resist[2] THEN
		 Cy_resist_2.xInit:=TRUE;
//	 END_IF
   //IF NOT Sensor_resist[3] THEN
		 Cy_resist_3.xInit:=TRUE;
//	 END_IF
 //  IF NOT Sensor_resist[4] THEN
		 Cy_resist_4.xInit:=TRUE;
//	 END_IF
 IF Cy_resist_1.xHP_Delay AND Cy_resist_2.xHP_Delay AND Cy_resist_3.xHP_Delay AND Cy_resist_4.xHP_Delay THEN
	     station.iStepInit := 30 ;	
 END_IF
 30://真空复位
      Va_ppu_1.xVacuumAuto := 
      Va_ppu_1.xVacuumManual := 
      Va_ppu_2.xVacuumAuto := 
      Va_ppu_2.xVacuumManual := FALSE ;
     	station.iStepInit:=40;
 40://轴上使能
    	Axis_PPU.xPowerInit := TRUE ;
    IF 	Axis_PPU.xPowerOn THEN 
    		station.iStepInit:=50;	
		END_IF		
50://轴回原点
    Axis_PPU.xHomeAuto := TRUE ;
		IF Axis_PPU.xHomeDone THEN
    Axis_PPU.xHomeAuto := FALSE ;
    		station.iStepInit:=60;	
		END_IF
60://轴去待机位
    Axis_PPU.xMoveAuto[1] := TRUE ;
		IF Axis_PPU.xMoveInPos[1] THEN 
    		station.iStepInit:=999;	
		END_IF	
 
 

			
999://初始化完成	
	station.iStepInit:=0;
	station.xInitDone:=TRUE;  
END_CASE
END_IF
END_ACTION

ACTION General:
 IF Machine_IO.xAutoMode   THEN //自动模式下
	 IF station.xRunning THEN
        //一轨 1 2
			//	IF CESHI THEN
	       IF NOT Sensor_resist[1] AND  Cy_resist_1.xHP_Delay THEN
			   Box_blow[1]:=FALSE;         //振动盘到前阻挡
				 ELSE
			   Box_blow[1]:=TRUE;					 
         END_IF
	       IF NOT Sensor_resist[2] AND  Cy_resist_2.xHP_Delay AND Sensor_resist[1] THEN
			   Cy_resist_1.xAuto:=TRUE;     //前阻挡到后阻挡
				 resist_open[1]    :=TRUE;
				 ELSE
				 resist_open[1]    :=FALSE;
				 IF  arTon[4].Q THEN
			   Cy_resist_1.xAuto:=FALSE;		
         END_IF			 
         END_IF	
	       IF arTon[1].Q  AND Sensor_resist[2] THEN
			   Cy_resist_2.xAuto:=TRUE;     //后阻挡到取料位
				 resist_open[2]    :=TRUE;
				 ELSE
				 resist_open[2]    :=FALSE;
				 IF  arTon[5].Q THEN
			   Cy_resist_2.xAuto:=FALSE;		
         END_IF					 
         END_IF	

				 
        //二轨 3  4
	       IF NOT Sensor_resist[3] AND  Cy_resist_3.xHP_Delay THEN
			   Box_blow[2]:=FALSE;         //振动盘到前阻挡
				 ELSE
			   Box_blow[2]:=TRUE;					 
         END_IF
	       IF NOT Sensor_resist[4] AND  Cy_resist_4.xHP_Delay AND Sensor_resist[3] THEN
			   Cy_resist_3.xAuto:=TRUE;     //前阻挡到后阻挡
				 resist_open[3]    :=TRUE;
				 ELSE
				 resist_open[3]    :=FALSE;
				 IF  arTon[6].Q THEN
			   Cy_resist_3.xAuto:=FALSE;		
         END_IF					 
         END_IF		
	       IF arTon[2].Q  AND Sensor_resist[4] THEN
			   Cy_resist_4.xAuto:=TRUE;     //后阻挡到取料位
				 resist_open[4]    :=TRUE;
				 ELSE
				 resist_open[4]    :=FALSE;
				 IF  arTon[7].Q THEN
			   Cy_resist_4.xAuto:=FALSE;		
         END_IF					 
         END_IF		
    IF NOT(Sensor_resist[1] AND  Sensor_resist[2] AND Sensor_resist[3] AND  Sensor_resist[4] AND  Sensor_cv_on[1] AND  Sensor_cv_on[2]) 
      THEN
		 Motion_S02_cv_run:=TRUE;//传送带运行置位
		 Box_run:=TRUE;	
		 ELSE
		 Motion_S02_cv_run:=FALSE;//传送带运行置位
		 Box_run:=FALSE	;			 
    END_IF 		 
   END_IF
END_IF
ft_cv(CLK:=station.xRunning OR CESHI , Q=> );//AND Machine_IO.xAutoMode
IF ft_cv.Q THEN
		 Motion_S02_cv_run:=FALSE;//传送带运行复位
		 Box_run:=FALSE;	 
		 Box_blow[1]:=FALSE;		
		 Box_blow[2]:=FALSE;		
 END_IF
//CT
rt_Ctmark(CLK:=Axis_PPU.xMoveInPos[1] , Q=>cycleTime.xCycleMark );

CT_DisAction_2[1](xCycleStartMark:=Axis_PPU.xMoveAuto[1] ,xCycleEndMark:=  Axis_PPU.xMoveInPos[1],xCycleRun:=TRUE, RCycleTime=>ct_show.S02_AXIS_POS1);
CT_DisAction_2[2](xCycleStartMark:=Axis_PPU.xMoveAuto[2] ,xCycleEndMark:=  Axis_PPU.xMoveInPos[2],xCycleRun:=TRUE, RCycleTime=>ct_show.S02_AXIS_POS2);
CT_DisAction_2[3](xCycleStartMark:=Axis_PPU.xMoveAuto[3] ,xCycleEndMark:=  Axis_PPU.xMoveInPos[3],xCycleRun:=TRUE, RCycleTime=>ct_show.S02_AXIS_POS3);
END_ACTION

ACTION ILC:

//---------------------------------------------------工站可执行-------------------------------------------------------
station.xCanRun := TRUE ;

//---------------------------------------------------气缸动作条件-------------------------------------------
Cy_resist_1.xOnILC:=
Cy_resist_1.xOffILC:=TRUE;

Cy_resist_2.xOnILC:=
Cy_resist_2.xOffILC:=TRUE;

Cy_resist_3.xOnILC:=
Cy_resist_3.xOffILC:=TRUE;

Cy_resist_4.xOnILC:=
Cy_resist_4.xOffILC:=TRUE;




//---------------------------------------------------伺服动作条件-------------------------------------------
	Axis_PPU.xJogILC :=     
	Axis_PPU.xHomeILC := 
	Axis_PPU.xRunILC := 
	Axis_PPU.xRelativeILC:=
	Axis_PPU.xMoveILC[1] :=                            //取料位
	Axis_PPU.xMoveILC[2] :=                            //放料位1
	Axis_PPU.xMoveILC[3] := TRUE;                      //放料位2
END_ACTION

ACTION TipAuto:

//------------------------------------------------AutoTip General---------------------------------


//------------------------------------------------AutoTip Cylinder--------------------------------

station.adwAutoTip[1].00:=FALSE;	//
station.adwAutoTip[1].01:=FALSE;	//
station.adwAutoTip[1].02:=Cy_resist_1.xAutoTip;	   //阻挡气缸1 气缸自动中有手动
station.adwAutoTip[1].03:=Cy_resist_2.xAutoTip;	   //阻挡气缸2 气缸自动中有手动
station.adwAutoTip[1].04:=Cy_resist_3.xAutoTip;	   //阻挡气缸3  气缸自动中有手动
station.adwAutoTip[1].05:=Cy_resist_4.xAutoTip;	   //阻挡气缸4 气缸自动中有手动
station.adwAutoTip[1].06:=FALSE;	   //真空1自动中有手动
station.adwAutoTip[1].07:=FALSE;	   //真空2自动中有手动

//伺服位置的读取,伺服位置错误自动提示               //Axis_distributor自动时位置错误
   FOR i:= 1 TO 5 BY 1 DO 
   	IF Axis_PPU.xMoveAuto[i] THEN
   		Axis_PPU.iPosNumber := i ;
   	END_IF
   END_FOR
IF fbMachine[1].xAutoMode AND NOT fbMachine[1].xRunning AND arTon_alarm[1].Q THEN 
	IF Axis_PPU.iPosNumber=1 AND NOT Axis_PPU.xMoveInPos[1] THEN station.adwAutoTip[1].08:=TRUE; END_IF //轴自动时位置不在位置1
	IF Axis_PPU.iPosNumber=2 AND NOT Axis_PPU.xMoveInPos[2] THEN station.adwAutoTip[1].09:=TRUE; END_IF //轴自动时位置不在位置2
	IF Axis_PPU.iPosNumber=3 AND NOT Axis_PPU.xMoveInPos[3] THEN station.adwAutoTip[1].10:=TRUE; END_IF //轴自动时位置不在位置3
END_IF
END_ACTION

END_PROGRAM

// Device/Application/POUS/02_STATION/S04_PushCard
PROGRAM S04_PushCard
VAR_INPUT
	//工站
	station					    : REFERENCE TO FB_Station:=fbStation[4];//工站状态
	cycleTime						: REFERENCE TO FB_CycleTime:= fbStCycleTime[4];	//工站CT
	//气缸
	Cy_lifter				    : REFERENCE TO FB_Cylinder:=fbCylinder[13];//推袋-升降
	Cy_push1				    : REFERENCE TO FB_Cylinder:=fbCylinder[14];//推袋1
	Cy_push2				    : REFERENCE TO FB_Cylinder:=fbCylinder[15];//推袋2




END_VAR
//内部变量
VAR
			arTon               :ARRAY[1..10] OF ton ;
      arTon_alarm           :ARRAY[1..10] OF ton ;  
	    rt_Ctmark           :R_TRIG;		
			CT_DisAction          : ARRAY[1..10] OF FB_CycleTime;
			CT_DisAction_1        : ARRAY[1..10] OF FB_CycleTime_1;			
	  	CT_DisAction_2        : ARRAY[1..10] OF FB_CycleTime_2;	
END_VAR

Alarm();
Delay();
FlowAuto();
FlowInit();
General();
ILC();
TipAuto();
TipManual();

ACTION Alarm:
station.adwAlarm[1].00:=station.xInitTimeout;	             //工站初始化超时报警
station.adwAlarm[1].01:=	Cy_push1.xHP_Off ;        
station.adwAlarm[1].02:=	Cy_push1.xWP_Off ;        
station.adwAlarm[1].03:=	Cy_push2.xHP_Off ;        //
station.adwAlarm[1].04:=	Cy_push2.xWP_Off ;        //
station.adwAlarm[1].05:=	Cy_lifter.xHP_Off ;        //
station.adwAlarm[1].06:=	Cy_lifter.xWP_Off ;        //
END_ACTION

ACTION Delay:

//----------------------------------------------动作延时-----------------------------------------------

arTon[1](IN:=   , PT:=T#10S , Q=> , ET=> );//
arTon[2](IN:=   , PT:=T#60S , Q=> , ET=> );//
arTon[3](IN:=   , PT:=T#60S , Q=> , ET=> );//
//----------------------------------------------报警延时-----------------------------------------------
arTon_alarm[1](IN:= , PT:=T#7S , Q=> , ET=> );//
arTon_alarm[2](IN:= , PT:=T#7S , Q=> , ET=> );//
arTon_alarm[3](IN:= , PT:=T#7S , Q=> , ET=> );//
arTon_alarm[4](IN:= , PT:=T#7S , Q=> , ET=> );//
arTon_alarm[5](IN:=   , PT:=T#60S , Q=> , ET=> );//
arTon_alarm[6](IN:=   , PT:=T#60S , Q=> , ET=> );//

arTon_alarm[7](IN:=   , PT:=T#10S , Q=> , ET=> );//
arTon_alarm[8](IN:=   , PT:=T#60S , Q=> , ET=> );//
arTon_alarm[9](IN:=   , PT:=T#60S , Q=> , ET=> );//
END_ACTION

ACTION FlowAuto:

//-----------------------------------------初始化是否完成判断----------------------------------------------
IF NOT station.xInitDone 
THEN
 	station.iStepAuto:=0;
 	station.xDone:=FALSE;
ELSIF station.xRunning 
THEN
//-----------------------------------------动作步骤--------------------------------------------------------
CASE station.iStepAuto OF	  
  	0: //----Home Step，等待启动----
		
		IF station.xDisabled AND station.xCanRun 	AND NOT fbMachine[1].xStopped AND NOT station.xSingleRunning 
		THEN
			station.xDone:=TRUE;//工站完成信号判断
		END_IF
		
	  IF  station.xSingleRunning OR station.xCanRun	AND NOT station.xDone AND NOT station.xDisabled	AND NOT fbMachine[1].xStopped
		THEN
			station.xCycleEnable:=TRUE;
			station.xDone:= FALSE;  
			station.iStepAuto:= 5;
		END_IF
		5://判断物料状态到位
      IF Axis_main_ready AND ((CardState[4].Card_OK AND BagState[3].Openbag_OK) OR station.xSingleRunFlag)// fbmachine[1].xTryRun)
        THEN
	//			Cy_lifter.xAuto:=TRUE;
	//			IF Cy_lifter.xHP_Delay THEN	
      			station.iStepAuto:= 10;
	//			END_IF
			END_IF
		10://推料	
		IF   Cy_push1.xHP_Delay AND CardState[4].A AND Axis_main_ready THEN
			Cy_push1.xAuto:=TRUE;
		END_IF
		IF   Cy_push2.xHP_Delay AND CardState[4].B AND Axis_main_ready THEN
			Cy_push2.xAuto:=TRUE;
		END_IF		
		
		IF  Cy_push1.xWP_Delay AND  Cy_push2.xWP_Delay  THEN
	    	CardState[4].Pushcard_OK:=TRUE;	
	      station.iStepAuto:= 20;
		END_IF		
		20://
					Cy_push2.xAuto:=FALSE;
		      Cy_push1.xAuto:=FALSE;
//					Cy_lifter.xAuto:=FALSE;
		IF  Cy_push1.xHP_Delay AND  Cy_push2.xHP_Delay  THEN	//AND Cy_lifter.xHP_Delay
	     	station.iStepAuto :=999;		
		END_IF
		 
		
		
	999://----Single Run Finish----
		station.xDone:=TRUE;
		station.xSingleRunFlag:=FALSE;
		station.xCycleEnable:=FALSE;	
    station.iStepAuto :=0;
END_CASE

END_IF
END_ACTION

ACTION FlowInit:
IF NOT station.xIniting THEN
  station.iStepInit:=0;    
ELSE
//--------------------------------------------初始化步序----------------------------------
CASE station.iStepInit OF	
 0://  
  	IF station.xIniting THEN	
  	  station.iStepInit:=10;	
  	END_IF	
10://复位数据
    
    station.iStepInit := 30 ;		
20://升降气缸原点
   Cy_lifter.xInit := TRUE ;
	  IF Cy_lifter.xHP_Delay   
   THEN 
    station.iStepInit:=30;	
		END_IF
30://气缸回原点
    Cy_push1.xInit := TRUE ;
    Cy_push2.xInit := TRUE ;
    IF Cy_push1.xHP_Delay AND Cy_push2.xHP_Delay 
     THEN 
    station.iStepInit:=999;	
		END_IF
		
999://初始化完成	
	station.iStepInit:=0;
	station.xInitDone:=TRUE;  
END_CASE
END_IF
END_ACTION

ACTION General:
//CT
rt_Ctmark(CLK:=station.xCycleEnable , Q=>cycleTime.xCycleMark );


CT_DisAction_2[1](xCycleStartMark:=Cy_push1.xHP_Valve ,xCycleEndMark:= Cy_push1.xHP_Delay,xCycleRun:=TRUE, RCycleTime=>ct_show.S04_Cy_push1_HP);
CT_DisAction_2[2](xCycleStartMark:=Cy_push1.xWP_Valve ,xCycleEndMark:= Cy_push1.xWP_Delay,xCycleRun:=TRUE, RCycleTime=>ct_show.S04_Cy_push1_WP);
CT_DisAction_2[3](xCycleStartMark:=Cy_push2.xHP_Valve ,xCycleEndMark:= Cy_push2.xHP_Delay,xCycleRun:=TRUE, RCycleTime=>ct_show.S04_Cy_push2_HP);
CT_DisAction_2[4](xCycleStartMark:=Cy_push2.xWP_Valve ,xCycleEndMark:= Cy_push2.xWP_Delay,xCycleRun:=TRUE, RCycleTime=>ct_show.S04_Cy_push2_WP);
END_ACTION

ACTION ILC:

//---------------------------------------------------工站可执行-------------------------------------------------------
station.xCanRun := TRUE ;

//---------------------------------------------------气缸动作条件-------------------------------------------
Cy_push1.xOnILC:=NOT S05_CircleLine.Axis_Cycleline.xbusy AND (S06_OpenBag.Cy_open.xHP_Sensor OR NOT S06_OpenBag.Axis_Y.xMoveInPos[2]);
Cy_push1.xOffILC:=TRUE;

Cy_push2.xOnILC:=NOT S05_CircleLine.Axis_Cycleline.xbusy AND (S06_OpenBag.Cy_open.xHP_Sensor OR NOT S06_OpenBag.Axis_Y.xMoveInPos[2]);
Cy_push2.xOffILC:=TRUE;

//Cy_lifter.xOnILC:=
//Cy_lifter.xOffILC:= TRUE;
END_ACTION

ACTION TipAuto:

//------------------------------------------------AutoTip General---------------------------------


//------------------------------------------------AutoTip Cylinder--------------------------------

station.adwAutoTip[1].00:=FALSE;	//
station.adwAutoTip[1].01:=FALSE;	//
station.adwAutoTip[1].02:=Cy_push1.xAutoTip;	       //Cy_push1 气缸自动中有手动
station.adwAutoTip[1].03:=Cy_push2.xAutoTip;	       //Cy_push2 气缸自动中有手动
//station.adwAutoTip[1].04:=Cy_lifter	.xAutoTip;	     //Cy_lifter 气缸自动中有手动
END_ACTION

ACTION TipManual:
//--------------------------------------------ManualTip------------------------------------------------------
station.adwManualTip[1].00			:=FALSE;//提示1
//-------------------------------------------气缸提示---------------------------------------------------------




/////////////////////////////////////////////////////////////////////////////////////////////////////////////////
END_ACTION

END_PROGRAM

// Device/Application/POUS/02_STATION/S06_OpenBag
PROGRAM S06_OpenBag
VAR_INPUT
	//工站
	station					    : REFERENCE TO FB_Station:=fbStation[6];//工站状态
	cycleTime						: REFERENCE TO FB_CycleTime:= fbStCycleTime[6];	//工站CT
   //伺服
   Axis_Y	          : REFERENCE TO FB_Axis:=fbAxis[3];
   //气缸
   	Cy_open				    : REFERENCE TO FB_Cylinder:=fbCylinder[12];//开袋
		Cy_lifter_HPSensor				   :BOOL;//升降
		Cy_lifter_Value              :BOOL;		
	//真空发生器
		Va_open_right				    : REFERENCE TO FB_Vacuum:=fbVacuum[5];     //张袋上真空
		Va_open_left			    : REFERENCE TO FB_Vacuum:=fbVacuum[6];     //张袋下真空


END_VAR
//内部变量
VAR
			arTon               :ARRAY[1..10] OF ton ; 
			arTon_alarm         :ARRAY[1..10] OF ton ; 
      rt_Ctmark           :R_TRIG;
			i                   :INT;
			CT_DisAction          : ARRAY[1..10] OF FB_CycleTime;
			CT_DisAction_1        : ARRAY[1..10] OF FB_CycleTime_1;			
	  	CT_DisAction_2        : ARRAY[1..10] OF FB_CycleTime_2;	
END_VAR

Alarm();
Delay();
FlowAuto();
FlowInit();
General();
ILC();
TipAuto();
TipManual();

ACTION Alarm:
station.adwAlarm[1].00:=station.xInitTimeout;	             //Add_distributor 工站初始化超时报警
//气缸
station.adwAlarm[1].01:=	Cy_open.xHP_Off ;        //
station.adwAlarm[1].02:=	Cy_open.xWP_Off ;        //
//真空
station.adwAlarm[1].03:=	Va_open_left.byAlarm.1;         //吸真空报警
station.adwAlarm[1].04:=	Va_open_left.byAlarm.3 ;        //破真空报警
station.adwAlarm[1].05:=	Va_open_right.byAlarm.1 ;        //
station.adwAlarm[1].06:=	Va_open_right.byAlarm.3 ;   
//轴
station.adwAlarm[1].07:=	  Axis_Y.xError ;             //轴报错
station.adwAlarm[1].08:=	  Axis_Y.xNotPowerOn;         //未使能
station.adwAlarm[1].09:=	  Axis_Y.xMoveTimeout;        //定位超时
END_ACTION

ACTION Delay:

//----------------------------------------------动作延时-----------------------------------------------

arTon[1](IN:= ((Va_open_left.xVacuumDelay OR NOT CardState[3].A)  AND ( Va_open_right.xVacuumDelay OR NOT CardState[3].B) OR fbmachine[1].xTryRun ) AND  station.iStepAuto=20 , PT:=T#100MS , Q=> , ET=> );////吸真空延时
arTon[2](IN:=NOT (Va_open_left.xVacuumDelay OR Va_open_right.xVacuumDelay) AND station.iStepAuto=40 , PT:=T#100MS , Q=> , ET=> );//破真空延时
arTon[3](IN:=  , PT:=T#1S , Q=> , ET=> );//
arTon[4](IN:=   , PT:=T#60S , Q=> , ET=> );//
arTon[5](IN:=   , PT:=T#60S , Q=> , ET=> );//
arTon[6](IN:=   , PT:=T#60S , Q=> , ET=> );//
//----------------------------------------------报警延时-----------------------------------------------
arTon_alarm[1](IN:=NOT Axis_Y.xbusy  , PT:=T#1S , Q=> , ET=> );//
arTon_alarm[2](IN:= , PT:=T#7S , Q=> , ET=> );//
arTon_alarm[3](IN:= , PT:=T#7S , Q=> , ET=> );//
arTon_alarm[4](IN:= , PT:=T#7S , Q=> , ET=> );//
arTon_alarm[5](IN:=   , PT:=T#60S , Q=> , ET=> );//
arTon_alarm[6](IN:=   , PT:=T#60S , Q=> , ET=> );//

arTon_alarm[7](IN:=   , PT:=T#10S , Q=> , ET=> );//
arTon_alarm[8](IN:=   , PT:=T#60S , Q=> , ET=> );//
arTon_alarm[9](IN:=   , PT:=T#60S , Q=> , ET=> );//
END_ACTION

ACTION FlowAuto:

//-----------------------------------------初始化是否完成判断----------------------------------------------
IF NOT station.xInitDone 
THEN
 	station.iStepAuto:=0;
 	station.xDone:=FALSE;
ELSIF station.xRunning  
THEN
//-----------------------------------------动作步骤--------------------------------------------------------
//POS1 取料位 POS2 放料位
//气缸原点：张开
CASE station.iStepAuto OF	  
	0: //----Home Step，等待启动----
		IF station.xDisabled AND station.xCanRun 	AND NOT fbMachine[1].xStopped AND NOT station.xSingleRunning 
		THEN
			station.xDone:=TRUE;//工站完成信号判断
		END_IF
		
	  IF  station.xSingleRunning OR station.xCanRun	AND NOT station.xDone AND NOT station.xDisabled	AND NOT fbMachine[1].xStopped
		THEN
			station.xCycleEnable:=TRUE;
			station.xDone:= FALSE;  
			station.iStepAuto:= 5;
		END_IF
	5://数据复位	
	  	Cy_lifter_Value := FALSE ;		
		  station.iStepAuto:= 10;
  10://	判断是否能张袋
	IF Cy_open.xHP_Delay  AND (NOT BagState[2].Suck_OK OR station.xSingleRunFlag) AND NOT S03_takebag.Axis_Cycleline.xbusy THEN 
		station.iStepAuto:= 11;
	END_IF			
  11:   
  IF  ( CardState[3].Card_OK OR station.xSingleRunFlag )AND NOT fbAxis[2].xbusy THEN      		 
      	station.iStepAuto:= 12;
	END_IF   
  12:                         								  
	IF NOT 	 Axis_Y.xMoveInPos[1]		THEN 		  								  
	 	Axis_Y.xMoveAuto[1] := TRUE ;
	END_IF	
	IF  Axis_Y.xMoveInPos[1] THEN 
			station.iStepAuto:= 15;
	END_IF	
	15://气缸闭合
   	Cy_open.xAuto:=TRUE;
		IF Cy_open.xWP_Delay THEN
	    station.iStepAuto:= 20;
		END_IF
  20://吸袋
     IF  NOT fbmachine[1].xTryRun THEN
        IF CardState[3].A THEN
	        	Va_open_left.xVacuumAuto:=TRUE;
       	END_IF
				IF CardState[3].B THEN
		        Va_open_right.xVacuumAuto:=TRUE;					
				END_IF
     END_IF
	IF arTon[1].Q THEN
			station.iStepAuto:= 25;
	END_IF
	25://先张开，再移动
	   	Cy_open.xAuto:=FALSE;
		IF Cy_open.xHP_Delay THEN
		 BagState[2].Suck_OK:=TRUE;//张袋完成
	   station.iStepAuto:= 30;
		END_IF	
  30://移到放料位
 //   Cy_open.xAuto:=FALSE;
  IF S03_takebag.Axis_Cycleline.xbusy OR station.xSingleRunFlag THEN
	 	Axis_Y.xMoveAuto[2] := TRUE ;
 END_IF
 		IF  Axis_Y.xMoveInPos[2] THEN 
		station.iStepAuto:= 40;
		END_IF	;
  40://破真空

	IF CardState[4].Pushcard_OK  OR station.xSingleRunFlag THEN 
 		Va_open_left.xVacuumAuto:=FALSE;
 		Va_open_right.xVacuumAuto:=FALSE;
		Cy_lifter_Value := TRUE ;
			IF arTon[2].Q THEN
		station.iStepAuto:= 50;
	END_IF
	END_IF

 50://回到取料位
   
	 	Axis_Y.xMoveAuto[1] := TRUE ;
		IF  Axis_Y.xMoveInPos[1] THEN 
		Cy_lifter_Value := FALSE ;
		station.iStepAuto:= 999;
		END_IF	;
	
		
	999://----Single Run Finish----
			
		station.iStepAuto :=0;
	//	station.xDone:=TRUE;
		station.xSingleRunFlag:=FALSE;
		station.xCycleEnable:=FALSE;	
END_CASE

END_IF
END_ACTION

ACTION FlowInit:
IF NOT station.xIniting THEN
  station.iStepInit:=0;    
ELSE
//--------------------------------------------初始化步序----------------------------------
CASE station.iStepInit OF	
 0://  
  	IF station.xIniting THEN	
  	  station.iStepInit:=10;	
  	END_IF	
10://复位数据
    BagState[2].Suck_OK:=FALSE;
    station.iStepInit := 20 ;		
20://真空复位
			Va_open_left.xVacuumAuto:=
			Va_open_left.xBreakAuto:=
			Va_open_left.xVacuumManual:=
			Va_open_right.xVacuumAuto:=
			Va_open_right.xBreakAuto:=
			Va_open_right.xVacuumManual:=FALSE;
			station.iStepInit:=30;	
 30://气缸
       Cy_open.xInit := TRUE ;
		   IF Cy_open.xHP_Delay   
       THEN 
        station.iStepInit:=35;	
		   END_IF
 35://新增压紧气缸
       Cy_lifter_Value := FALSE ;
		   IF Cy_lifter_HPSensor  
       THEN 
        station.iStepInit:=40;	
		   END_IF			 
 40://轴上使能
    
			Axis_Y.xPowerInit := TRUE ;
    IF  Axis_Y.xPowerOn THEN 
    		station.iStepInit:=60;	
		END_IF		
50://轴回原点
   
    Axis_Y.xHomeAuto := TRUE ;
		IF   Axis_Y.xHomeDone THEN
    
		    Axis_Y.xHomeAuto := FALSE ;
    		station.iStepInit:=60;	
		END_IF
60://轴去待机位
   
	  Axis_Y.xMoveAuto[1] := TRUE ;
		IF  Axis_Y.xMoveInPos[1] THEN 
    		station.iStepInit:=999;	
		END_IF	
 
 

			
999://初始化完成	
	station.iStepInit:=0;
	station.xInitDone:=TRUE;  
END_CASE
END_IF
END_ACTION

ACTION General:

//空跑屏蔽真空发生器
Va_open_left.xAlarmDisable:= 
Va_open_right.xAlarmDisable:= fbmachine[1].xTryRun;

//CT

CT_DisAction_2[1](xCycleStartMark:=Axis_Y.xMoveAuto[1] ,xCycleEndMark:=  Axis_Y.xMoveInPos[1],xCycleRun:=TRUE, RCycleTime=>ct_show.S06_AXIS_POS1);
CT_DisAction_2[2](xCycleStartMark:=Axis_Y.xMoveAuto[2] ,xCycleEndMark:=  Axis_Y.xMoveInPos[2],xCycleRun:=TRUE, RCycleTime=>ct_show.S06_AXIS_POS2);
CT_DisAction_2[3](xCycleStartMark:=Cy_open.xHP_Valve ,xCycleEndMark:= Cy_open.xHP_Delay,xCycleRun:=TRUE, RCycleTime=>ct_show.S06_Cy_open_HP);
CT_DisAction_2[4](xCycleStartMark:=Cy_open.xWP_Valve ,xCycleEndMark:= Cy_open.xWP_Delay,xCycleRun:=TRUE, RCycleTime=>ct_show.S06_Cy_open_WP);
//Openbag_OK
IF (Cy_open.xHP_Delay AND Axis_Y.xMoveInPos[2]  AND fbStation[6].iStepAuto = 40) OR station.xDisabled  THEN  
	BagState[3].Openbag_OK:=TRUE; 
	ELSE
	BagState[3].Openbag_OK:=FALSE;
END_IF
END_ACTION

ACTION ILC:

//---------------------------------------------------工站可执行-------------------------------------------------------
station.xCanRun := TRUE ;

//---------------------------------------------------气缸动作条件-------------------------------------------
Cy_open.xOnILC:=
Cy_open.xOffILC:=TRUE;








//---------------------------------------------------伺服动作条件-------------------------------------------

	
	Axis_Y.xJogILC :=     
	Axis_Y.xHomeILC := 
	Axis_Y.xRunILC := 
	Axis_Y.xRelativeILC:= 
	Axis_Y.xMoveILC[1] :=                            //取料位
	Axis_Y.xMoveILC[2] :=                            //放料位1
	Axis_Y.xMoveILC[3] :=  TRUE ;                      //放料位2
END_ACTION

ACTION TipAuto:

//------------------------------------------------AutoTip General---------------------------------


//------------------------------------------------AutoTip Cylinder--------------------------------

station.adwAutoTip[1].00:=FALSE;	//
station.adwAutoTip[1].01:=FALSE;	//

station.adwAutoTip[1].02:=Cy_open.xAutoTip;	   //开袋气缸自动中有手动
station.adwAutoTip[1].03:=FALSE;	   //左真空自动中有手动
station.adwAutoTip[1].04:=FALSE;	   //右真空自动中有手动
//伺服位置的读取,伺服位置错误自动提示               //Axis_distributor自动时位置错误
   FOR i:= 1 TO 5 BY 1 DO 
   	IF Axis_Y.xMoveAuto[i] THEN
   		Axis_Y.iPosNumber := i ;
   	END_IF
   END_FOR
IF fbMachine[1].xAutoMode AND NOT fbMachine[1].xRunning AND arTon_alarm[1].Q THEN 
	IF Axis_Y.iPosNumber=1 AND NOT Axis_Y.xMoveInPos[1] THEN station.adwAutoTip[1].08:=TRUE; END_IF //轴自动时位置不在位置1
	IF Axis_Y.iPosNumber=2 AND NOT Axis_Y.xMoveInPos[2] THEN station.adwAutoTip[1].09:=TRUE; END_IF //轴自动时位置不在位置2
	IF Axis_Y.iPosNumber=3 AND NOT Axis_Y.xMoveInPos[3] THEN station.adwAutoTip[1].10:=TRUE; END_IF //轴自动时位置不在位置3
END_IF
END_ACTION

ACTION TipManual:
//--------------------------------------------ManualTip------------------------------------------------------
station.adwManualTip[1].00			:=FALSE;//提示1
//-------------------------------------------气缸提示---------------------------------------------------------




/////////////////////////////////////////////////////////////////////////////////////////////////////////////////
END_ACTION

END_PROGRAM

// Device/Application/POUS/01_LINK/OUTPUT
PROGRAM OUTPUT
VAR
END_VAR

//-----------------------------------模块一-----------------------------------------------
Output_local[1].channel_1.0 :=Machine_IO.xStartLight;
Output_local[1].channel_1.1 :=Machine_IO.xStopLight;
Output_local[1].channel_1.2 :=Machine_IO.xResetLight;
Output_local[1].channel_1.3 :=Machine_IO.xInitLight;
//Output_local[1].channel_1.4 :=
Output_local[1].channel_1.5 :=Machine_IO.xTriLightYellow  := fbMachine[1].xLampYellow; 
Output_local[1].channel_1.6 :=Machine_IO.xTriLightGreen   := fbMachine[1].xLampGreen;
Output_local[1].channel_1.7 :=Machine_IO.xTriLightRed     :=fbMachine[1].xLampRed;

Output_local[1].channel_2.0 :=Machine_IO.xBuzzer          := fbMachine[1].xLampBuzzer;
//Output_local[1].channel_2.1 :=Add_distributor.Cy_takeClamp1_1.xHP_Valve;
Output_local[1].channel_2.2 :=Add_distributor.Cy_takeClamp1_1.xWP_Valve; //分料夹爪气缸一拖6
(*Output_local[1].channel_2.3 :=Add_distributor.Cy_takeClamp1_2.xHP_Valve;
Output_local[1].channel_2.4 :=Add_distributor.Cy_takeClamp1_2.xWP_Valve;
Output_local[1].channel_2.5 :=Add_distributor.Cy_takeClamp2_1.xHP_Valve;
Output_local[1].channel_2.6 :=Add_distributor.Cy_takeClamp2_1.xWP_Valve;
Output_local[1].channel_2.7 :=Add_distributor.Cy_takeClamp2_2.xHP_Valve;

Output_local[1].channel_3.0 :=Add_distributor.Cy_takeClamp2_2.xWP_Valve;
Output_local[1].channel_3.1 :=Add_distributor.Cy_takeClamp3_1.xHP_Valve;
Output_local[1].channel_3.2 :=Add_distributor.Cy_takeClamp3_1.xWP_Valve;
Output_local[1].channel_3.3 :=Add_distributor.Cy_takeClamp3_2.xHP_Valve;
Output_local[1].channel_3.4 :=Add_distributor.Cy_takeClamp3_2.xWP_Valve;
*)
//Output_local[1].channel_3.5 :=Add_distributor.Cy_openleft.xHP_Valve;
Output_local[1].channel_3.6 :=Add_distributor.Cy_openleft.xWP_Valve;//单控阀
//Output_local[1].channel_3.7 :=Add_distributor.Cy_openright.xHP_Valve;

Output_local[1].channel_4.0 :=Add_distributor.Cy_openright.xWP_Valve;//单控阀
Output_local[1].channel_4.1 :=Add_distributor.Cy_lifter.xHP_Valve;
Output_local[1].channel_4.2 :=Add_distributor.Cy_lifter.xWP_Valve;
//Output_local[1].channel_4.3 :=
//Output_local[1].channel_4.4 :=
//Output_local[1].channel_4.5 :=
//Output_local[1].channel_4.6 :=
//Output_local[1].channel_4.7 :=

//-----------------------------------模块二-----------------------------------------------
//Output_local[2].channel_1.0 :=S01_transplant.Cy_rotate.xHP_Valve;
Output_local[2].channel_1.1 :=S01_transplant.Cy_rotate.xWP_Valve;        //单控阀
//Output_local[2].channel_1.2 :=S01_transplant.Cy_takeClamp1.xHP_Valve;
Output_local[2].channel_1.3 :=S01_transplant.Cy_takeClamp1.xWP_Valve;    //单控阀
//Output_local[2].channel_1.4 :=S01_transplant.Cy_takeClamp2.xHP_Valve;
//Output_local[2].channel_1.5 :=S01_transplant.Cy_takeClamp2.xWP_Valve;
//Output_local[2].channel_1.6 :=S01_transplant.Cy_takeClamp3.xHP_Valve;
Output_local[2].channel_1.7 :=S01_transplant.Cy_takeClamp3.xWP_Valve;    //单控阀

//Output_local[2].channel_2.0 :=S01_transplant.Cy_takeClamp4.xHP_Valve;
//Output_local[2].channel_2.1 :=S01_transplant.Cy_takeClamp4.xWP_Valve;
Output_local[2].channel_2.2 :=S01_transplant.Cy_lifter.xHP_Valve;
Output_local[2].channel_2.3 :=S01_transplant.Cy_lifter.xWP_Valve;
//Output_local[2].channel_2.4 :=
//Output_local[2].channel_2.5 :=
//Output_local[2].channel_2.6 :=
//Output_local[2].channel_2.7 :=

Output_local[2].channel_3.0 :=S02_bowlFeeder.Cy_resist_1.xHP_Valve;
Output_local[2].channel_3.1 :=S02_bowlFeeder.Cy_resist_1.xWP_Valve;
Output_local[2].channel_3.2 :=S02_bowlFeeder.Cy_resist_2.xHP_Valve;
Output_local[2].channel_3.3 :=S02_bowlFeeder.Cy_resist_2.xWP_Valve;
Output_local[2].channel_3.4 :=S02_bowlFeeder.Cy_resist_3.xHP_Valve;
Output_local[2].channel_3.5 :=S02_bowlFeeder.Cy_resist_3.xWP_Valve;
Output_local[2].channel_3.6 :=S02_bowlFeeder.Cy_resist_4.xHP_Valve;
Output_local[2].channel_3.7 :=S02_bowlFeeder.Cy_resist_4.xWP_Valve;

Output_local[2].channel_4.0 :=Motion_ADD_cv_run[1];
Output_local[2].channel_4.1 :=Motion_ADD_cv_run[2];
Output_local[2].channel_4.2 :=Motion_S02_cv_run;
//Output_local[2].channel_4.3 :=
//Output_local[2].channel_4.4 :=
//Output_local[2].channel_4.5 :=
//Output_local[2].channel_4.6 :=
//Output_local[2].channel_4.7 :=

//-----------------------------------模块三-----------------------------------------------
Output_local[3].channel_1.0 :=S02_bowlFeeder.Va_ppu_1.xVacuumValve;
Output_local[3].channel_1.1 :=S02_bowlFeeder.Va_ppu_1.xBreakValve;
Output_local[3].channel_1.2 :=S02_bowlFeeder.Va_ppu_2.xVacuumValve;
Output_local[3].channel_1.3 :=S02_bowlFeeder.Va_ppu_2.xBreakValve;
//Output_local[3].channel_1.4 :=
//Output_local[3].channel_1.5 :=
//Output_local[3].channel_1.6 :=
//Output_local[3].channel_1.7 :=

//Output_local[3].channel_2.0 :=S03_takebag.Cy_lifter.xHP_Valve;
Output_local[3].channel_2.1 :=S03_takebag.Cy_lifter.xWP_Valve;
Output_local[3].channel_2.2 :=S03_takebag.Va_take1.xVacuumValve;
//Output_local[3].channel_2.3 :=S03_takebag.Va_take1.xBreakValve;
Output_local[3].channel_2.4 :=S03_takebag.Va_take2.xVacuumValve;
//Output_local[3].channel_2.5 :=S03_takebag.Va_take2.xBreakValve;
//Output_local[3].channel_2.6 :=S06_packcard.Cy_open.xHP_Valve;
Output_local[3].channel_2.7 :=S06_OpenBag.Cy_open.xWP_Valve;

Output_local[3].channel_3.0 :=S06_OpenBag.Va_open_left.xVacuumValve;
//Output_local[3].channel_3.1 :=S06_packcard.Va_open_left.xBreakValve;
Output_local[3].channel_3.2 :=S06_OpenBag.Va_open_right.xVacuumValve;
//Output_local[3].channel_3.3 :=S06_packcard.Va_open_right.xBreakValve;
Output_local[3].channel_3.4 :=Box_blow[1];
Output_local[3].channel_3.5 :=Box_blow[2];
Output_local[3].channel_3.6 :=Box_run;
//Output_local[3].channel_3.7 :=

//Output_local[3].channel_4.0 :=S04_bagging.Cy_lifter.xHP_Valve;
Output_local[3].channel_4.1 :=S04_PushCard.Cy_lifter.xWP_Valve;
//Output_local[3].channel_4.2 :=S04_bagging.Cy_push1.xHP_Valve;
Output_local[3].channel_4.3 :=S04_PushCard.Cy_push1.xWP_Valve;
//Output_local[3].channel_4.4 :=S04_bagging.Cy_push2.xHP_Valve;
Output_local[3].channel_4.5 :=S04_PushCard.Cy_push2.xWP_Valve;
//Output_local[3].channel_4.6 :=
//Output_local[3].channel_4.7 :=

END_PROGRAM

// Device/Application/POUS/03_CALL_standard/CallStandard
PROGRAM CallStandard
VAR_INPUT
	{attribute 'hide'}
	fbBlinker					: ARRAY[1..10] OF FB_Blinker;//自定义脉冲发生功能块
	bWindowColseHmi             : ARRAY[1..5]OF BOOL ; //窗口关闭
END_VAR
VAR
   Run,_firstSMC,_firstJD,_firstRGI41,_firstPerPump,_firstEPSRobot,_firstInjectPump,_firstCentrifuge	: BOOL;
	 bCylinder_First,bStation_First,bVacuum_First,bStation_First1,bMachine_First,bMachine_First1 : BOOL ;
	 i,j,k,t,nIndex : INT ;
	arAlarm: INT;
	ton100ms : TON ;
	_xMotorRunning : BOOL ;
	_ton1 : TON ;
	_xPower1 , _xPower2 : BOOL := TRUE;;
	_xButtonSMC,_xButtonCentrifuge : BOOL ;

	
	GVL_HMI_Temp: INT;
	uSafeDoor   :UINT;
END_VAR

ACT_Blink();
ACT_CT();
ACT_Cylinder();
ACT_Machine();
ACT_Proface();
ACT_Station();
ACT_Vacuum();

ACTION ACT_Cylinder:
//上电复位
IF NOT bCylinder_First THEN
  FOR j :=1 TO gc_uiCylinderNum DO 
  fbCylinder[j].xHmi               :=FALSE;	   //复位HMI上的按钮
  END_FOR
  bCylinder_First                :=TRUE;
END_IF


FOR i:=1 TO gc_uiCylinderNum DO
fbCylinder[i](
	xEStop:=fbMachine[1].xEStop,  
	xSafety:=fbMachine[1].xSafety , 
	xManualMode:=fbMachine[1].xManualMode , 
	xAutoMode:=fbMachine[1].xAutoMode , 
	xAirOn:=fbMachine[1].xAirOn , 
	tAlarm:= , 
	xReset:=fbMachine[1].xReset , 
	xAlarmDisable:= , 
	xHmi:= , 
	tHP_Delay:=INT_TO_TIME(stData.Cy_Pers[i].iHP_Delay) , 
	tWP_Delay:=INT_TO_TIME(stData.Cy_Pers[i].iHP_Delay) ,  
	xHP_Valve=> , 
	xWP_Valve=> , 
	xHP_Delay=> , 
	xWP_Delay=> );
END_FOR
END_ACTION

ACTION ACT_Machine:


FOR nIndex:=1 TO gc_uiMachineNum DO
fbMachine[nIndex](
	xEmptyHmi:= , 
	xTryRun:= , 
	xEmptyConfirmHmi:= , 
	xInitConfirm:= ,
  xStart:=  fbProface[1].xStartHmi  OR  Machine_IO.xStartButton,//HMI+实体按钮
  xStop:=   fbProface[1].xStopHmi OR Machine_IO.xStopButton ,
  xReset:=  fbProface[1].xResetHmi OR Machine_IO.xResetButton ,
  xPause:=  fbProface[1].xPauseHmi OR Machine_IO.xStopButton ,
  xInit:=   fbProface[1].xInitHmi  OR Machine_IO.xInitButton,
  xManualMode:= Machine_IO.xManualMode ,
  xAutoMode:= Machine_IO.xAutoMode ,	 
	xDoorClosed := (uSafeDoor=16) OR  HMI_Other.xShieldSafetyDoor,
	xEStop := Machine_IO.xEstopButton[1] AND Machine_IO.xEstopButton[2] ,		   
  xKey := TRUE,
  xAirOn := Machine_IO.xAiron,
  xShieldBuzzzer :=  HMI_Other.xShieldBuzzer ,
  xSafety:=fbMachine[1].xDoorClosed 
						AND fbMachine[1].xEStop 
						AND fbMachine[1].xAirOn 
						AND fbMachine[1].xKey ,
	xRunning=>  , 
	xEmptying=> ,
	xEStopped=> , 
	xIniting=>  , 
	diCycleTime => ,
	xStopped=> , 
	xPaused=> , 	
   );
	 
	END_FOR

// 读取保存的生产数据
IF NOT bMachine_First THEN
   FOR i:=1 TO gc_uiMachineNum BY 1 DO 
   	fbMachine[i].udiGoods := MachinePers[i].udiGoods ;
   	fbMachine[i].udiBads  := MachinePers[i].udiBads ;
   	fbMachine[i].udiTotal := MachinePers[i].udiTotal ;
   	fbMachine[i].rReject  := MachinePers[i].rReject ;
   	fbMachine[i].rYield   := MachinePers[i].rYield ;	
   END_FOR
    bMachine_First := TRUE ;
END_IF
//将生产数据写给HMI
IF 	stSysPulse.xP100ms THEN
   FOR i:=1 TO gc_uiMachineNum BY 1 DO 
   MachinePers[i].udiGoods := fbMachine[i].udiGoods ;
   MachinePers[i].udiBads 	  := fbMachine[i].udiBads ; 
   MachinePers[i].udiTotal	  := fbMachine[i].udiTotal ;
   MachinePers[i].rReject 	  := fbMachine[i].rReject ; 
   MachinePers[i].rYield     := fbMachine[i].rYield ;  
   END_FOR
END_IF 
uSafeDoor:=0;
FOR i:=1 TO 16 BY 1 DO
	IF Machine_IO.xSafeDoor[i] THEN
		uSafeDoor:=uSafeDoor+1;
	END_IF
END_FOR
END_ACTION

ACTION ACT_Station:
//上电复位
IF NOT bStation_First THEN
  FOR t :=1 TO gc_uiStationNum DO 
    fbStation[t].xCycleRunHmi:=FALSE;
    fbStation[t].xInitHmi:=FALSE;
    fbStation[t].xJogRunHmi:=FALSE;
    fbStation[t].xPauseHmi:=FALSE;
  END_FOR
  bStation_First:=TRUE;
END_IF

FOR k:=1 TO gc_uiStationNum DO
	fbStation[k](
		xEStop:=fbMachine[1].xEStop , 
		xKey:=fbMachine[1].xKey , 
		xSafety:=fbMachine[1].xSafety , 
		xManualMode:=fbMachine[1].xManualMode , 
		xReset:=fbMachine[1].xReset , 
		xMachinePause:=fbMachine[1].xPause , 
		xMachineReInit:=fbMachine[1].xReInit , 
		xMachineIniting:=fbMachine[1].xIniting , 
		xMachineRunning:=fbMachine[1].xRunning , 
		tInitTimeout:= , 
		xInitHmi:= , 
		xInitDone:= , 
		xDisabled:= , 
		xCycleRunHmi:= , 
		xJogRunHmi:= , 
		xPauseHmi:= , 
		xCycleRunning=> , 
		xJogRunning=> , 
		xSingleRunning=> , 
		xRunning=> , 
		uiState=> , 
		diCycleTime =>   
	);

END_FOR
END_ACTION

ACTION ACT_Proface:
fbProface[1](                                              //
	xEStop									:=fbMachine[1].xEStop,
	xSafety									:=fbMachine[1].xSafety,
	xManualMode							:=fbMachine[1].xManualMode,
	xAutoMode								:=fbMachine[1].xAutoMode,
	xAlarm									:=fbMachine[1].xAlarm,
	xTip										:=fbMachine[1].xTip,
	xInit										:=fbMachine[1].xInit,
	xIniting								:=fbMachine[1].xIniting,
	xInitDone								:=fbMachine[1].xInitDone,
	xDummyCheckDone					:=fbMachine[1].xDummyDone,
	xEmptyDone							:=fbMachine[1].xEmptyDone,
);
END_ACTION

ACTION ACT_Blink:

//	生成特定周期的振荡矩形波，可用于指示灯的闪烁，不可用于精确计时
fbBlinker[1](
	tBlink:=T#10MS,
	bBlink=>stSysPulse.xP10ms,
	brBlink=>stSysPulse.xR10ms,
	bfBlink=>stSysPulse.xF10ms
);
fbBlinker[2](
	tBlink:=T#20MS,
	bBlink=>stSysPulse.xP20ms,
	brBlink=>stSysPulse.xR20ms,
	bfBlink=>stSysPulse.xF20ms
);
fbBlinker[3](
	tBlink:=T#50MS,
	bBlink=>stSysPulse.xP50ms,
	brBlink=>stSysPulse.xR50ms,
	bfBlink=>stSysPulse.xF50ms
);
fbBlinker[4](
	tBlink:=T#100MS,
	bBlink=>stSysPulse.xP100ms,
	brBlink=>stSysPulse.xR100ms,
	bfBlink=>stSysPulse.xF100ms
);
fbBlinker[5](
	tBlink:=T#200MS,
	bBlink=>stSysPulse.xP200ms,
	brBlink=>stSysPulse.xR200ms,
	bfBlink=>stSysPulse.xF200ms
);
fbBlinker[6](
	tBlink:=T#500MS,
	bBlink=>stSysPulse.xP500ms,
	brBlink=>stSysPulse.xR500ms,
	bfBlink=>stSysPulse.xF500ms
);
fbBlinker[7](
	tBlink:=T#1S,
	bBlink=>stSysPulse.xP1s,
	brBlink=>stSysPulse.xR1s,
	bfBlink=>stSysPulse.xF1s
);
fbBlinker[8](
	tBlink:=T#2S,
	bBlink=>stSysPulse.xP2s,
	brBlink=>stSysPulse.xR2s,
	bfBlink=>stSysPulse.xF2s
);
fbBlinker[9](
	tBlink:=T#5S,
	bBlink=>stSysPulse.xP5s,
	brBlink=>stSysPulse.xR5s,
	bfBlink=>stSysPulse.xF5s
);
fbBlinker[10](
	tBlink:=T#10S,
	bBlink=>stSysPulse.xP10s,
	brBlink=>stSysPulse.xR10s,
	bfBlink=>stSysPulse.xF10s
);
END_ACTION

ACTION ACT_Vacuum:
//上电复位
IF NOT bVacuum_First THEN
  FOR t :=1 TO gc_uiVacuumNum DO 
      fbVacuum[t].xVacuumHmi:=
      fbVacuum[t].xBreakHmi:=FALSE;
  END_FOR
  bVacuum_First:=TRUE;
END_IF

FOR nIndex:=1 TO gc_uiVacuumNum DO
	fbVacuum[nIndex](
	    xManualMode:=fbMachine[1].xManualMode , 
	    xAirOn:=fbMachine[1].xAirOn , 
	    xReset:=fbMachine[1].xReset , 
	    xAlarmDisable:= , 
	    xVacuumHmi:= , 
	    xBreakHmi:= , 
	    tBreakDelay:=INT_TO_TIME(stData.Vac_Pers[nIndex].iBreakDelay) , 
	    tVacuumDelay:=INT_TO_TIME(stData.Vac_Pers[nIndex].iVacuumDelay) , 
	    xVacuumValve=> , 
	    xBreakValve=> , 
	    xVacuumDelay=> , 
	    xBreakDelay=> , 
	    byAlarm=> );
END_FOR
END_ACTION

ACTION ACT_CT:
FOR k:=1 TO gc_uiStationNum BY 1 DO
	fbStCycleTime[k]
  (xCycleMark:= , 
   xCycleRun:= TRUE, 
   rCycleTime=> );
END_FOR
END_ACTION

END_PROGRAM

// Device/Application/FB/12_BlinkFB/FB_Blinker
FUNCTION_BLOCK FB_Blinker
VAR_INPUT
	tBlink						: TIME;					//脉冲宽度
END_VAR

VAR_OUTPUT
	bBlink						: BOOL;					//输出脉冲
	brBlink						: BOOL;					//输出脉冲上升沿
	bfBlink						: BOOL;					//输出脉冲上升沿
END_VAR

VAR
	 
	tonBlink					: TON;					//计时
	{attribute 'hide'}
	 
	rtBlink						: R_TRIG;				//脉冲上升沿
	 {attribute 'hide'}
	ftBlink						: F_TRIG;				//脉冲下降沿
	{attribute 'hide'}
END_VAR

tonBlink(
	IN:=NOT tonBlink.Q,
	PT:=tBlink / 2,
	Q=>);
IF tonBlink.Q THEN
	bBlink:=NOT bBlink;
END_IF

rtBlink(CLK:=bBlink, Q=>brBlink);
ftBlink(CLK:=bBlink, Q=>bfBlink);

END_FUNCTION_BLOCK

// Device/Application/POUS/03_CALL_standard/ControlMachine
PROGRAM ControlMachine
VAR
	_ftrigTryRun : f_trig ;//空跑按钮下降沿
	ft_outcountA:    F_TRIG;
	ft_outcountB:    F_TRIG;	
	T_ECState       :TON;
	xAlarm                      	: BOOL;
	xWarning											: BOOL;
END_VAR

ACT_ALarm();
ACT_Count();
ACT_Try_run();
ACT_InitDone();

ACTION ACT_Try_run:
//空跑标识位用的输入。。结束后需要工站重新初始化
_ftrigTryRun(CLK:= fbmachine[1].xTryRun , Q=> );
IF  _ftrigTryRun.Q THEN 
	FOR K:=1 TO  gc_uiStationNum	BY 1 DO
	IF 		fbStation[K].iStepAuto <> 0 THEN
		fbStation[K].xInitDone:=FALSE;
	END_IF
	END_FOR
END_IF
END_ACTION

ACTION ACT_Count:
//计数
ft_outcountA(CLK:= BagState[3].Loose_OK  , Q=> );
IF ft_outcountA.Q THEN
	fbMachine[1].udiGoods:=fbMachine[1].udiGoods+1;
END_IF
IF ft_outcountB.Q THEN
	fbMachine[1].udiGoods:=fbMachine[1].udiGoods+1;
END_IF
IF HMI_Other.xOutCountZero THEN
fbMachine[1].udiGoods:=0;//---作为出料数量
END_IF
//fbMachine[1].udiTotal:=;//----作为进料数量
END_ACTION

ACTION ACT_ALarm:
//--------------------------------------------Machine alarm------------------------------------------------

//----机台状态提示----

fbMachine[1].dwMessage[1].00			:=	fbMachine[1].xRunning;			//设备自动中
fbMachine[1].dwMessage[1].01		  :=	fbMachine[1].xStopped;			//设备停止状态
fbMachine[1].dwMessage[1].02			:=	fbMachine[1].xPaused;			//设备暂停状态
fbMachine[1].dwMessage[1].03			:=	fbMachine[1].xAlarm;			//设备报警中
fbMachine[1].dwMessage[1].04			:=	fbMachine[1].xIniting;			//设备初始化中
fbMachine[1].dwMessage[1].05			:=	fbMachine[1].xEmptying;			//设备清料中

//----机台报警信息----

//光栅遮挡报警

//安全门被打开
IF NOT HMI_Other.xShieldSafetyDoor THEN
IF fbMachine[1].xAutoMode AND NOT Machine_IO.xSafeDoor[1]  THEN fbMachine[1].dwAlarm[1].00:=TRUE; END_IF	//[M01.00] 设备安全门1被打开
IF fbMachine[1].xAutoMode AND NOT Machine_IO.xSafeDoor[2]  THEN fbMachine[1].dwAlarm[1].01:=TRUE; END_IF	//[M01.1 ] 设备安全门2 被打开
IF fbMachine[1].xAutoMode AND NOT Machine_IO.xSafeDoor[3]  THEN fbMachine[1].dwAlarm[1].02:=TRUE; END_IF	//[M01.2 ] 设备安全门3 被打开
IF fbMachine[1].xAutoMode AND NOT Machine_IO.xSafeDoor[4]  THEN fbMachine[1].dwAlarm[1].03:=TRUE; END_IF	//[M01.3 ] 设备安全门4 被打开
IF fbMachine[1].xAutoMode AND NOT Machine_IO.xSafeDoor[5]  THEN fbMachine[1].dwAlarm[1].04:=TRUE; END_IF	//[M01.4 ] 设备安全门5 被打开
IF fbMachine[1].xAutoMode AND NOT Machine_IO.xSafeDoor[6]  THEN fbMachine[1].dwAlarm[1].05:=TRUE; END_IF	//[M01.5 ] 设备安全门6 被打开
IF fbMachine[1].xAutoMode AND NOT Machine_IO.xSafeDoor[7]  THEN fbMachine[1].dwAlarm[1].06:=TRUE; END_IF	//[M01.6 ] 设备安全门7 被打开
IF fbMachine[1].xAutoMode AND NOT Machine_IO.xSafeDoor[8]  THEN fbMachine[1].dwAlarm[1].07:=TRUE; END_IF	//[M01.7 ] 设备安全门8 被打开
IF fbMachine[1].xAutoMode AND NOT Machine_IO.xSafeDoor[9]  THEN fbMachine[1].dwAlarm[1].08:=TRUE; END_IF	//[M01.8 ] 设备安全门9 被打开
IF fbMachine[1].xAutoMode AND NOT Machine_IO.xSafeDoor[10] THEN fbMachine[1].dwAlarm[1].09:=TRUE; END_IF	//[M01.9 ] 设备安全门10 被打开
IF fbMachine[1].xAutoMode AND NOT Machine_IO.xSafeDoor[11] THEN fbMachine[1].dwAlarm[1].10:=TRUE; END_IF	//[M01.10] 设备安全门11被打开
IF fbMachine[1].xAutoMode AND NOT Machine_IO.xSafeDoor[12] THEN fbMachine[1].dwAlarm[1].11:=TRUE; END_IF	//[M01.11] 设备安全门12被打开
IF fbMachine[1].xAutoMode AND NOT Machine_IO.xSafeDoor[13] THEN fbMachine[1].dwAlarm[1].12:=TRUE; END_IF	//[M01.12] 设备安全门13被打开
IF fbMachine[1].xAutoMode AND NOT Machine_IO.xSafeDoor[14] THEN fbMachine[1].dwAlarm[1].13:=TRUE; END_IF	//[M01.13] 设备安全门14被打开
IF fbMachine[1].xAutoMode AND NOT Machine_IO.xSafeDoor[15] THEN fbMachine[1].dwAlarm[1].14:=TRUE; END_IF	//[M01.14] 设备安全门15被打开
IF fbMachine[1].xAutoMode AND NOT Machine_IO.xSafeDoor[16] THEN fbMachine[1].dwAlarm[1].15:=TRUE; END_IF	//[M01.15] 设备安全门16被打开
END_IF
//气源异常
IF NOT fbMachine[1].xAirOn THEN
	fbMachine[1].dwAlarm[1].16:=TRUE; //[M01.16] 设备气压报警
END_IF
//急停被按下
IF NOT Machine_IO.xEstopButton[1]   THEN fbMachine[1].dwAlarm[1].17:=TRUE; END_IF //[M01.17] 设备急停00被按下
IF NOT Machine_IO.xEstopButton[2]   THEN fbMachine[1].dwAlarm[1].18:=TRUE; END_IF //[M01.18] 设备急停1 被按下
//EC总线异常
T_ECState(IN:=NOT EthercatStatus.xProRunStatus AND NOT fbMachine[1].xReset, PT:=T#5S , Q=> , ET=> );//
IF T_ECState.Q THEN
	fbMachine[1].dwAlarm[1].19:=TRUE;
END_IF
//----工站报警汇总----

xAlarm:= FALSE;							//先复位
FOR K :=1 TO gc_uiStationNum DO 
  IF fbStation[K].xAlarm THEN		//整机故障单独 
    xAlarm:=TRUE; 
  END_IF
END_FOR

//----机台报警----
fbMachine[1].xAlarm:=
  fbMachine[1].dwAlarm[1]<>0
	OR fbMachine[1].dwAlarm[2]<>0
	OR fbMachine[1].dwAlarm[3]<>0
	OR fbMachine[1].dwAlarm[4]<>0
	OR fbMachine[1].dwAlarm[5]<>0
	OR xAlarm;
END_ACTION

ACTION ACT_InitDone:

//------------------------------------------------初始化完成汇总-------------------------------------


//------------------------------------------------初始化完成汇总-------------------------------------
fbMachine[1].xInitDone:=TRUE;//先置位
FOR K:=1 TO gc_uiStationNum DO 
  IF NOT fbStation[K].xInitDone
  THEN 
    fbMachine[1].xInitDone:=FALSE; 
  END_IF
END_FOR
END_ACTION

END_PROGRAM

// Device/Application/POUS/03_CALL_standard/Call_Axis
PROGRAM Call_Axis
VAR
	arrayMoveFalse : ARRAY[1..gc_uiAxisMoveNum] OF BOOL ;//给HMI去位置指令复位
	K : INT;//索引
END_VAR

ACT_Check();
ACT_Link();

ACTION ACT_Link:

//------------------------------------------上电第一个扫描周期操作-------------------------------------------
IF  EthercatStatus.xFirstCycle  THEN
	
	RealAxis[1].Server                  :=ADR(S01_CycleLine);
    RealAxis[1].Axis                    :=ADR(Axis_2); //产品传送带
		
	RealAxis[2].Server                  :=ADR(S03_CycleLine);
    RealAxis[2].Axis                    :=ADR(Axis_3); //供袋传送带	
		
		
	RealAxis[3].Server                  :=ADR(S03_supplybag_Y);
    RealAxis[3].Axis                    :=ADR(Axis_4); //供袋张口轴---横移
		
	RealAxis[4].Server                  :=ADR(S02_PPU_Module);
    RealAxis[4].Axis                    :=ADR(Axis_5); //PPU模组，取干燥剂
		
	RealAxis[5].Server                  :=ADR(Add_distributor_Y);//
    RealAxis[5].Axis                    :=ADR(Axis_1);//分料轴---3变4
				
END_IF

IF EthercatStatus.xFirstCycle THEN
  FOR K :=1 TO (gc_uiAxisNum) DO 
      fbAxis[K].xAlarmResetHmi                   :=     			   //HMI_故障复位
	    fbAxis[K].xPowerHmi                        :=     			   //HMI_使能
	    fbAxis[K].xJogForwardHmi                   :=     			   //HMI_正点
	    fbAxis[K].xJogBackwardsHmi                 :=     			   //HMI_反点
	    fbAxis[K].xHomeHmi                         :=     			   //HMI_回零
	    fbAxis[K].xStopHmi                         :=FALSE;			   //HMI_停止
	    fbAxis[K].xMoveHmi                         :=arrayMoveFalse;   //HMI_轴启动
		//给轴空参数赋值
		IF 	stData.Axis[K].rJogVelocity	<=0 THEN
		stData.Axis[K].rJogVelocity				:=20;		
		END_IF
		IF stData.Axis[K].rManualVelocity<=0 THEN
		stData.Axis[K].rManualVelocity				:=50;	
		END_IF
		IF stData.Axis[K].rAutoVelocity<=0 THEN
		stData.Axis[K].rAutoVelocity			    :=100;
		END_IF
		IF stData.Axis[K].rJogAcceleration<=0 THEN
		stData.Axis[K].rJogAcceleration            :=50; 
		END_IF
		IF stData.Axis[K].rJogDeceleration<=0 THEN
		stData.Axis[K].rJogDeceleration            :=50; 
		END_IF
		IF  stData.Axis[K].rVelocityAcc<=0 THEN
		stData.Axis[K].rVelocityAcc                :=50; 
		END_IF
		IF stData.Axis[K].rVelocityDec<=0 THEN
		stData.Axis[K].rVelocityDec                :=50; 
		END_IF
		IF stData.Axis[K].rMoveAcceleration<=0 THEN
		stData.Axis[K].rMoveAcceleration           :=2000; 
		END_IF
		IF stData.Axis[K].rMoveDeceleration<=0 THEN
		stData.Axis[K].rMoveDeceleration           :=2000;  
		END_IF
  END_FOR                                       			
END_IF
//------------------------------------------轴控功能块调用-------------------------------------------	
//----伺服----
IF EthercatStatus.xProRunStatus 
THEN
  	FOR K:=1 TO (gc_uiAxisNum) DO
fbAxis[K](
	Basic_Axis:=RealAxis[K] , 
	xEStop:=fbMachine[1].xEStop , 
	xKey:=fbMachine[1].xKey , 
	xSafety:=fbMachine[1].xSafety ,                                          //安全条件：门、急停、气源等
	xManualMode:=fbMachine[1].xManualMode AND NOT fbMachine[1].xIniting ,    //手动模式
	xAutoMode:=fbMachine[1].xRunning OR fbMachine[1].xIniting ,              //自动模式
	xReset:=fbMachine[1].xReset  , 
	xStopHmi:= , 
	xPowerHmi:= , 
	xBrakeHmi:= , 
	xHomeHmi:= , 
	xAlarmResetHmi:= , 
	xJogForwardHmi:= , 
	xJogBackwardsHmi:=  , 
	xMoveHmi:= , 
	xRelativeHmi:= , 
	rJogAcceleration:=  stData.Axis[K].rJogAcceleration, 
	rJogDeceleration:=  stData.Axis[K].rJogDeceleration , 
	rMoveAcceleration:= stData.Axis[K].rMoveAcceleration , 
	rMoveDeceleration:= stData.Axis[K].rMoveDeceleration , 
	rJogVelocity:=      stData.Axis[K].rJogVelocity , 
	rManualVelocity:=   stData.Axis[K].rManualVelocity , 
	rAutoVelocity:=     stData.Axis[K].rAutoVelocity , 
	rMovePosition:=     stData.Axis[K].rMovePosition , 
	rMoveVelocity:=     stData.Axis[K].rMoveVelocity , 
	rRelativeDistance:= stData.Axis[K].rRelativeDistance , 
	rRelativeVelocity:= stData.Axis[K].rRelativeVelocity , 
	rVelocityVel:=      stData.Axis[K].rVelocityVel , 
	rVelocityAcc:=      stData.Axis[K].rJogAcceleration , 
	rVelocityDec:=      stData.Axis[K].rJogDeceleration , 
	xPowerOn=> , 
	xBrakeUnlock=> , 
	xReady=> , 
	xHomeDone=> , 
	xMoveInPos=> , 
	xRelativeDone1=> , 
	xError=> , 
	udiErrorID=> , 
	rActTorque=> , 
	rActPos=> , 
	rActVelo=> , 
  );
  END_FOR	

END_IF
stData.Axis[3].rAutoVelocity:=stData.Axis[2].rAutoVelocity:=stData.Axis[1].rAutoVelocity;
stData.Axis[3].rMoveAcceleration:=stData.Axis[2].rMoveAcceleration:=stData.Axis[1].rMoveAcceleration;
stData.Axis[3].rMoveDeceleration:=stData.Axis[2].rMoveDeceleration:=stData.Axis[1].rMoveDeceleration;
END_ACTION

ACTION ACT_Check:
//----------------------------------------EtherCAT网络检测--------------------------------------

EthercatStatus.xEtherCAT_OK:=ETHERCAT.xConfigFinished AND ETHERCAT.xDistributedClockInSync AND NOT ETHERCAT.xError;//系统判断EC网络OK
EthercatStatus.xFirstCycle      :=EthercatStatus.xEtherCAT_OK AND NOT EthercatStatus.xProRunStatus  ;//EC网络OK,第一个循环绑一次轴
EthercatStatus.xProRunStatus      :=EthercatStatus.xFirstCycle OR EthercatStatus.xProRunStatus;//EC网络OK后常通

//---------------------------------------如果报错，一直复位网络-----------------------------------
IF ETHERCAT.xError THEN
	ETHERCAT.xRestart:=TRUE;
ELSE
	ETHERCAT.xRestart:=FALSE;
END_IF
//---------------------------------------
END_ACTION

END_PROGRAM

// Device/Application/FB/14_MachineFB/FB_Machine
FUNCTION_BLOCK FB_Machine
VAR_INPUT
	xEStop						: BOOL;					//急停(运行时常ON)
	xKey						: BOOL;					//钥匙开关
	xDoorClosed					: BOOL;					//所有安全门关好
	xSafety						: BOOL;					//安全防护中
	xAirOn						: BOOL;					//气压正常
	xAlarm						: BOOL;					//报警中
	xManualTip					: BOOL;					//手动提示中
	xAutoTip					: BOOL;					//自动提示中
	xTip						: BOOL;					//提示中
	xShieldBuzzzer :BOOL;       //蜂鸣器屏蔽
	
	xStart						: BOOL;					//启动按钮
	xStop						: BOOL;					//停止按钮
	xReset						: BOOL;					//复位按钮
	xPause						: BOOL;					//暂停按钮
	xInit						: BOOL;					//初始化按钮
	xManualMode					: BOOL;					//手动模式
	xAutoMode					: BOOL;					//自动模式

	
	xInitConfirm				: BOOL;					//初始化确认
	xInitDone					: BOOL;					//初始化完成
	tInitTimeout				: TIME:=T#3M;			//初始化超时延时
	
	xDummyMode					: BOOL;					//点检模式，点检使能
	xStationDummyDone			: BOOL;					//工站点检完成
	xDummyDone					: BOOL;					//点检完成
	xDummyDoneConfirm			: BOOL;					//点检完成确认
	
	xSampling					: BOOL;					//取样中
	uiSampleCount				: UINT;					//取样数量统计
	xSampleDone					: BOOL;					//取样完成
	xEmptyHmi					: BOOL;					//清料HMI
	xEmptyConfirmHmi			: BOOL;					//清料确认HMI
	xEmptyDone					: BOOL;					//清料完成
	xOrderFinished				: BOOL;					//订单完成
	xOrderChanged				: BOOL;					//订单切换
	
	xTryRun						: BOOL;					//空跑试运行
	xCycleEnable      	 		: BOOL;          		//设备CT计时
	xDataEmpty					: BOOL;					//数据清空
	tDataEmpty					: TIME;					//数据清空延时，默认为0
	xCarrierDataClear			: BOOL;					//载座数据清空
	tCarrierDataClear			: TIME;					//载座数据清空延时，默认为0
	
	xInitConfirmDialog			: BOOL;					//初始化确认对话框
	
	dwStatus					:ARRAY[1..4] OF DWORD;	//状态，bit.0急停中.1钥匙关闭.2气压低.3手动模式.4自动模式.5未准备好.6准备就绪.7运行中.8停止中.9报警中.10暂停中.11初始化中.12清料中.13清料完成.14取样中.15取样完成.16订单完成.17点检屏蔽中.18要求点检.其它可自定义	
 
	dwMessage					:ARRAY[1..5] OF DWORD;	//提示信息
	dwAlarm						:ARRAY[1..5] OF DWORD;	//报警信息	
	
	xDummyDisabled				: REFERENCE TO BOOL;	//点检屏
	//rCycleTime				: REAL;					//生产周期，单位s
	//生产信息相关变量
	udiGoods					: UDINT;				//当前良品数量
	udiBads						: UDINT;				//当前不良数量
	udiTotal					:  UDINT;				//当前总数量
	rYield						:  REAL;				//当前良品率
	rReject						:  REAL;				//当前不良率
END_VAR

VAR_OUTPUT
	xEStopped					: BOOL;					//急停状态
	xRunning					: BOOL;					//自动中
	xStopped					: BOOL;					//停止状态
	xPaused						: BOOL;					//暂停状态
	xIniting					: BOOL;					//初始化中
	xEmptying					: BOOL;					//清料中
	
	xAutoModeTip				: BOOL;					//自动模式上升沿提示
	
	xInitTimeout				: BOOL;					//初始化超时
	xReInit						: BOOL;					//整机重新初始化，用于复位各工站初始化完成
	
	xInitDoneDialog				: BOOL;					//初始化完成对话框
	xInitFailedDialog			: BOOL;					//初始化失败对话框
	
	xEmptyConfirmDialog			: BOOL;					//清料确认对话框
	xEmptyDoneDialog			: BOOL;					//清料完成对话框
	
	xShowAlarm					: BOOL;					//报警信息显示
	xShowTip					: BOOL;					//提示信息显示
	
	xStartLight					: BOOL;					//启动按钮灯
	xStopLight					: BOOL;					//停止按钮灯
	xResetLight					: BOOL;					//复位按钮灯
	xPauseLight					: BOOL;					//暂停按钮灯
	xInitLight					: BOOL;					//初始化按钮灯
	
	xLampGreen					: BOOL;					//三色灯-绿
	xLampYellow					: BOOL;					//三色灯-黄
	xLampRed					: BOOL;					//三色灯-红
	xLampBuzzer					: BOOL;					//三色灯-蜂鸣器	
	
	diCycleTime        			: DINT;					//基础时间是100ms

END_VAR

VAR
	{attribute 'hide'}
	rtRunning					: R_TRIG;				//自动中上升沿
	{attribute 'hide'}
	rtEmptyDone					: R_TRIG;				//清料完成上升沿
	{attribute 'hide'}
	tonDataEmpty				: TON;					//数据清零延时
	rtDataEmpty					: R_TRIG;				//数据清空上升沿
	{attribute 'hide'}
	tonCarrierDataClear			: TON;					//载座数据清空延时
	rtCarrierDataClear			: R_TRIG;				//载座数据清空上升沿
	{attribute 'hide'}
	xDummyWarnTime				: BOOL;					//点检提醒时间
	{attribute 'hide'}
	rtDummyWarnTime				: R_TRIG;				//点检提醒时间上升沿
	{attribute 'hide'}
	xDummyAlarmTime				: BOOL;					//点检报警时间
	{attribute 'hide'}
	rtDummyAlarmTime			: R_TRIG;				//点检报警时间上升沿
	{attribute 'hide'}
	rtDummyDoneConfirm			: R_TRIG;				//点检完成确认上升沿
	{attribute 'hide'}
	xDummyDoneCache				: BOOL;					//点检完成缓存
	{attribute 'hide'}
	xDummyComplete				: BOOL;					//点检完成状态
	{attribute 'hide'}
	xDummyRequirement			: BOOL;					//要求点检提醒
	{attribute 'hide'}
	rtInit						: R_TRIG;				//初始化上升沿
	{attribute 'hide'}
	rtInitConfirm				: R_TRIG;				//初始化确认上升沿
	{attribute 'hide'}
	ftIniting					: F_TRIG;				//初始化下降沿
	{attribute 'hide'}
	rtEmptyHmi					: R_TRIG;				//清料HMI上升沿
	{attribute 'hide'}
	ftEmptying					: F_TRIG;				//清料中下降沿
	{attribute 'hide'}
	xInitAble					: BOOL;					//初始化条件
	{attribute 'hide'}
	xRunAble					: BOOL;					//运行条件
	{attribute 'hide'}
	tonInitTimeout				: TON;					//初始化超时
	{attribute 'hide'}
	tonLampBuzzer				: TON;					//蜂鸣器关闭延时
	{attribute 'hide'}
	rtCycleFlag					: R_TRIG;				//循环标志上升沿
	{attribute 'hide'}
	lrCycleTimer				: LREAL;				//计时器，单位100ns，除于10000后单位ms
	{attribute 'hide'}
	tonHydraGoodsOut			: TON;					//Hydra良品输出信号延时
	{attribute 'hide'}
	tonHydraGoodsInterval		: TON;					//Hydra良品输出信号间隔
	{attribute 'hide'}
	tonHydraBadsOut				: TON;					//Hydra不良输出信号延时
	{attribute 'hide'}
	tonHydraBadsInterval		: TON;					//Hydra不良输出信号间隔
	
	rtAutoMode					: R_TRIG;				//自动模式上升沿
	rMachineStart       		: R_TRIG;
	i : INT ;

END_VAR

ACT_General();
ACT_Init();
ACT_Empty();
ACT_Start();
ACT_Pause();
ACT_Stop();
ACT_Reset();
ACT_Lamp();
ACT_Data();
ACT_CycleTime();

ACTION ACT_Stop:
//	停止中
IF xStop AND xRunning THEN
	xStopped:=TRUE;
END_IF

IF xEStopped
	OR xStart
	OR xPaused
THEN
	xStopped:=FALSE;
END_IF

//停止按钮灯，停止中常亮
xStopLight:=xStopped;
END_ACTION

ACTION ACT_Data:
//	当前数据清零
tonDataEmpty(IN:=xDataEmpty, PT:=tDataEmpty, Q=> , ET=> );
rtDataEmpty(CLK:=tonDataEmpty.Q, Q=> );
IF rtDataEmpty.Q THEN
	udiGoods:=0;
	udiBads:=0;
END_IF

//	计算当前良品率
udiTotal:=udiGoods + udiBads;
IF udiTotal > 0 THEN
	rYield:=LREAL_TO_REAL(100 * UDINT_TO_LREAL(udiGoods) / UDINT_TO_LREAL(udiTotal));
	rReject:=100.0 - rYield;
ELSE
	rReject:=0;
	rYield:=0;
END_IF



//	转台数据清零上升沿
tonCarrierDataClear(IN:=xCarrierDataClear, PT:=tCarrierDataClear, Q=> , ET=> );
rtCarrierDataClear(CLK:=tonCarrierDataClear.Q, Q=> );
END_ACTION

ACTION ACT_Empty:
//	启动时，先复位清料完成
IF xStart
	AND NOT xRunning
	AND NOT xEmptying
THEN
	xEmptyDone:=FALSE;
END_IF

//	清料HMI上升沿，弹出清料确认对话框
rtEmptyHmi(CLK:=xEmptyHmi, Q=> );
xEmptyConfirmDialog:=rtEmptyHmi.Q
	AND xEStop
	AND xKey
	AND xSafety
	AND xInitDone
	AND NOT xAlarm
	AND NOT xTip
	AND NOT xIniting;

//	清料
IF xEStop
	AND NOT xIniting
	AND NOT xEmptyDone
THEN
	IF xEmptyConfirmHmi
		AND xKey
		AND xSafety
		AND xInitDone
		AND NOT xAlarm
		AND NOT xTip
	THEN
		xEmptying:=TRUE;
	END_IF
ELSE
	xEmptying:=FALSE;
END_IF

//	清料中下降沿，弹出清料完成对话框
ftEmptying(CLK:=xEmptying, Q=> );
xEmptyDoneDialog:=ftEmptying.Q
	AND xEmptyDone;
END_ACTION

ACTION ACT_General:
//	急停中
xEStopped:=NOT xEStop;

xShowAlarm := FALSE;
FOR i:=1 TO 4 BY 1 DO 	
 IF dwMessage[i]<>0 THEN 
		xShowAlarm := TRUE ;
		EXIT ;
 END_IF
END_FOR
//提示报警显示
xShowAlarm:= xShowAlarm OR xAlarm;

//提示信息显示
xShowTip:=xTip;

//报警复位
IF xReset THEN
	FOR i:=1 TO 5 BY 1 DO 
		dwMessage[i] := dwAlarm[i]  := 0;
	END_FOR
END_IF
END_ACTION

ACTION ACT_Init:
//	初始化条件
xInitAble:=xEStop
	AND xKey
	AND xSafety
	AND xManualMode
	AND NOT xAlarm
	AND NOT xInitTimeout;

//	初始化上升沿，弹出初始化确认对话框
rtInit(CLK:=xInit, Q=> );
IF rtInit.Q AND xInitAble AND NOT xIniting THEN
  xInitConfirmDialog :=TRUE;	
END_IF
(*bInitConfirmDialog:=rtInit.Q
	AND bInitAble
	AND NOT bIniting;*)

//	初始化确认上升沿，触发各工站重新初始化
rtInitConfirm(CLK:=xInitConfirm, Q=> );
xReInit:=rtInitConfirm.Q
	AND xInitAble
	AND NOT xIniting;
//false初始化弹出的窗口
IF rtInitConfirm.Q
THEN 
  xInitConfirmDialog :=FALSE;
  
END_IF

//	初始化中
IF xInitAble
	AND NOT xPause
	AND NOT xInitDone
THEN
	IF xInitConfirm THEN
		xIniting:=TRUE;
	END_IF
ELSE
	xIniting:=FALSE;
END_IF

//	初始化按钮灯，初始化中闪烁，初始化完成熄灭
xInitLight:=xIniting AND stSysPulse.xP1s ;

//	初始化超时
tonInitTimeout(
	IN:=xIniting,
	PT:=tInitTimeout,
	Q=> , ET=>
);
IF xReset THEN
	xInitTimeout:=FALSE;
END_IF
IF tonInitTimeout.Q THEN
	xInitTimeout:=TRUE;
END_IF

//	初始化中下降沿，弹出初始化完成或失败对话框
ftIniting(CLK:=xIniting, Q=> );
xInitDoneDialog:=ftIniting.Q
	AND xInitDone;
xInitFailedDialog:=ftIniting.Q
	AND NOT xInitDone;
END_ACTION

ACTION ACT_Lamp:
//	三色灯-绿，运行中绿灯常亮
xLampGreen:=xRunning;

//	三色灯-红，报警或急停中红灯常亮
xLampRed:=xAlarm OR xEStopped;

//	三色灯-黄，其余情况下黄灯常亮，有等待信息时黄灯闪烁

xLampYellow:=NOT xLampGreen AND NOT xLampRed AND stSysPulse.xP1s;	

//	蜂鸣器关闭延时
tonLampBuzzer(IN:=xAlarm, PT:=T#3S, Q=> , ET=> );

//	三色灯-蜂鸣器
xLampBuzzer:=xAlarm
	AND stSysPulse.xP1s
	AND NOT tonLampBuzzer.Q
	AND NOT xShieldBuzzzer;
END_ACTION

ACTION ACT_Pause:
//	暂停中
IF xPause  THEN
	xPaused:=TRUE;
END_IF

IF xEStopped
	OR xStart
THEN
	xPaused:=FALSE;
END_IF

//暂停按钮灯，暂停中常亮
xPauseLight:=xPaused;
END_ACTION

ACTION ACT_Reset:
//	复位按钮灯，报警时闪烁
xResetLight:=xAlarm
	AND stSysPulse.xP1s;
END_ACTION

ACTION ACT_Start:
//	运行条件
xRunAble:=xEStop
	AND xKey
	AND xSafety
	AND xAutoMode
	AND xInitDone
	AND NOT xAlarm
	AND NOT xAutoTip
	AND NOT xStopped;

//	运行中
IF xRunAble
	AND NOT xPause
	AND NOT xEmptyDone//清料完成
THEN
	IF xStart THEN
		xRunning:=TRUE;
	END_IF
ELSE
	xRunning:=FALSE;
END_IF

//	启动按钮灯，运行中常亮，准备就绪时闪烁
xStartLight:=xRunning
	OR xRunAble
		AND stSysPulse.xP1s;
END_ACTION

ACTION ACT_CycleTime:
//	初始化时同时初始化工站周期计时
IF xIniting THEN
	xCycleEnable:=FALSE;
END_IF

//工站完成触发信号
rMachineStart(CLK:= xCycleEnable);
IF rMachineStart.Q
THEN
	diCycleTime := 0;
END_IF
//	工站周期计时
IF xRunning AND xCycleEnable AND stSysPulse.xR100ms
THEN
	diCycleTime := diCycleTime + 1;//对应最小周期是0.1ms
END_IF
END_ACTION

END_FUNCTION_BLOCK

// Device/Application/FB/17_HMIFB/FB_Proface
FUNCTION_BLOCK FB_Proface
VAR_INPUT
	xEStop								: BOOL;					//急停
	xSafety								: BOOL;					//安全防护
	xManualMode							: BOOL;					//手动模式
	xAutoMode							: BOOL;					//自动模式
	xAlarm								: BOOL;					//报警中
	xTip								: BOOL;					//提示中
	xInit								: BOOL;					//初始化
	xIniting							: BOOL;					//初始化中
	xInitDone							: BOOL;					//初始化完成
	xDummyChecking						: BOOL;					//点检中
	xDummyCheckDone						: BOOL;					//点检完成
	xEmptying							: BOOL;					//清料中
	xEmptyDone							: BOOL;					//清料完成
	xStartHmi							: BOOL;					//启动HMI
	xStopHmi							: BOOL;					//停止HMI
	xResetHmi							: BOOL;					//复位HMI
	xPauseHmi							: BOOL;					//暂停HMI
	xInitHmi							: BOOL;					//初始化HMI
	xManualModeHmi						: BOOL;					//手动HMI
	xAutoModeHmi						: BOOL;					//自动HMI
	xUnlockHmi							: BOOL;					//解锁HMI
	xDummyCheckHmi						: BOOL;					//点检HMI
	xEmptyHmi							: BOOL;					//清料HMI
	xWindowColseHmi						: BOOL;					//窗口关闭HMI
	                      		
	nCurrentPageIndex					: UINT:=0;				//当前画面索引
	nJumpToPageIndex					: UINT:=1;				//跳转到画面索引
	                      		
	nWindowControlIndex					: UINT:=0;				//窗口控制索引
	nWindowNumberIndex					: UINT:=1;				//窗口编号索引
	nWindowLocationIndexX				: UINT:=2;				//窗口位置索引X坐标
	nWindowLocationIndexY				: UINT:=3;				//窗口位置索引Y坐标
	                      		
	nWindowLocationX					: UINT:=300;			//窗口位置X坐标
	nWindowLocationY					: UINT:=80;		    //窗口位置Y坐标
	                      		
	nInitConfirmWindow					: UINT:=1;				//初始化确认窗口编号
	nInitAlarmWindow					: UINT:=2;				//初始化有报警窗口编号
	nInitingAlarmWindow					: UINT:=3;				//初始化中有报警窗口编号
	nInitingWindow						: UINT:=4;				//初始化中窗口编号
	nInitDoneWindow						: UINT:=5;				//初始化完成窗口编号
	nInitFailWindow						: UINT:=6;				//初始化失败窗口编号
	
	nDummyCheckConfirmWindow			: UINT:=5;				//点检确认窗口编号
	nDummyCheckDoneWindow				: UINT:=6;				//点检完成窗口编号
	nDummyCheckFailWindow				: UINT:=7;				//点检失败窗口编号
	
	nEmptyConfirmWindow					: UINT:=10;				//清料确认窗口编号
	nEmptyDoneWindow					: UINT:=11;				//清料完成窗口编号
	
	nTipWindow							: UINT:=31;				//提示窗口编号
	nButtonWindow						: UINT:=121;			//调试窗口编号
END_VAR

VAR_OUTPUT
END_VAR

VAR
	
	xStartLight							: BOOL;					//启动灯
	xStopLight							: BOOL;					//停止灯
	xResetLight							: BOOL;					//复位灯
	xPauseLight							: BOOL;					//暂停灯
	xInitLight							: BOOL;					//初始化灯
	
END_VAR
VAR_INPUT
	wWindow								: ARRAY[0..20] OF WORD;	//窗口控制区	
END_VAR
VAR
	
	wSystem								: ARRAY[0..20] OF WORD;	//系统区

	                  				
	ftTip								: F_TRIG;				//提示中下降沿
	rtInit								: R_TRIG;				//初始化上升沿
	ftIniting							: F_TRIG;				//初始化中下降沿
	rtDummyCheck						: R_TRIG;				//点检上升沿
	ftDummyChecking						: F_TRIG;				//点检中下降沿
	rtEmptyConfirm						: R_TRIG;				//清料确认上升沿
	rtEmptyDone							: R_TRIG;				//清料完成上升沿
	
END_VAR

ACT_Init();
ACT_DummyCheck();
ACT_Empty();
ACT_Control();

ACTION ACT_Control:
ftTip(CLK:=xTip, Q=>);
IF xWindowColseHMI		//窗口关闭
	OR ftTip.Q			//提示下降沿自动关闭窗口
THEN
	wWindow[nWindowNumberIndex]:=0;
END_IF

IF xTip THEN
	wWindow[nWindowNumberIndex]:=nTipWindow;
END_IF

wWindow[nWindowControlIndex].0:=wWindow[nWindowNumberIndex]<>0;

wWindow[nWindowLocationIndexX]:=nWindowLocationX;
wWindow[nWindowLocationIndexY]:=nWindowLocationY;
END_ACTION

ACTION ACT_Empty:
rtEmptyConfirm(CLK:=xEmptyHmi, Q=>);
rtEmptyDone(CLK:=xEmptyDone, Q=>);
IF rtEmptyConfirm.Q		//清料确认窗口显示
	AND fbMachine[1].xEStop
	AND fbMachine[1].xSafety
	AND fbMachine[1].xAutoMode
	AND fbMachine[1].xInitDone
	AND NOT fbMachine[1].xAlarm
THEN
	wWindow[nWindowNumberIndex]:=nEmptyConfirmWindow;
END_IF

IF rtEmptyDone.Q THEN	//清料完成窗口显示
	wWindow[nWindowNumberIndex]:=nEmptyDoneWindow;
END_IF
END_ACTION

ACTION ACT_DummyCheck:
rtDummyCheck(CLK:=xDummyCheckHmi, Q=>);
ftDummyChecking(CLK:=xDummyChecking, Q=>);
IF rtDummyCheck.Q	//点检确认窗口显示
	AND xEStop
	AND xSafety
	AND xManualMode
	AND xInitDone
	AND NOT xAlarm
THEN
	wWindow[nWindowNumberIndex]:=nDummyCheckConfirmWindow;
END_IF
IF ftDummyChecking.Q THEN
	IF xDummyCheckDone THEN		//点检完成窗口显示
		wWindow[nWindowNumberIndex]:=nDummyCheckDoneWindow;
	ELSE	//点检失败窗口显示
		wWindow[nWindowNumberIndex]:=nDummyCheckFailWindow;
	END_IF
END_IF
END_ACTION

ACTION ACT_Init:
rtInit(CLK:=xInit, Q=>);
ftIniting(CLK:=xIniting, Q=>);

IF rtInit.Q
THEN
	wSystem[0]:=10;
END_IF

IF rtInit.Q					//初始化确认窗口显示
	AND xEStop
	AND xSafety
	AND xManualMode
	AND NOT xAlarm
	AND NOT xIniting
THEN
	wWindow[nWindowNumberIndex]:=nInitConfirmWindow;
END_IF

IF rtInit.Q					//初始化有报警
	AND xAlarm
THEN
	wWindow[nWindowNumberIndex]:=nInitAlarmWindow;
END_IF

IF xIniting					//初始化中有报警
	AND xAlarm
THEN
	wWindow[nWindowNumberIndex]:=nInitingAlarmWindow;
END_IF

IF xIniting THEN			//初始化中窗口显示
	wWindow[nWindowNumberIndex]:=nInitingWindow;
END_IF

IF ftIniting.Q THEN		
	IF xInitDone THEN		//初始化完成窗口显示
		wWindow[nWindowNumberIndex]:=nInitDoneWindow;
	ELSE					//初始化失败窗口显示
		wWindow[nWindowNumberIndex]:=nInitFailWindow;
	END_IF
END_IF

IF xWindowColseHMI
THEN
	wWindow[nWindowNumberIndex]:=0;
	wWindow[nWindowControlIndex]:=0;
END_IF
END_ACTION

END_FUNCTION_BLOCK

// Device/Application/FB/14_MachineFB/FB_Machine_1
FUNCTION_BLOCK FB_Machine_1
VAR_INPUT
	CT_input           :BOOL;   //计时信号
	CT_number          :REAL:=1;//出料数量设定
	Sta_xtart_b        :BOOL;   //启动按钮
	Sta_xstop_b        :BOOL;   //停止按钮
	Sta_xreset_b       :BOOL;   //复位按钮
	Sta_safety         :BOOL;   //安全条件、
END_VAR
VAR_OUTPUT
	CT_TIME            :REAL;   //节拍时间
	Sta_xrunning       :BOOL;   //运行状态
	Sta_xstop          :BOOL;   //停止状态
	Sta_xiniting       :BOOL;   //初始化中
	Sta_xPaused        :BOOL;   //暂停中
	Sta_xEmptying      :BOOL;   //清料中（排空）
END_VAR
VAR_IN_OUT
END_VAR
VAR
	CT_Rtinput            : R_TRIG;         //计时信号上升沿
	CT_TEMP               : UDINT;
	CT_Start              : UDINT;
	CT_Stop               : UDINT;
END_VAR

ACTION ACT_CT:

//  CT计算
CT_Rtinput(CLK:= CT_input , Q=> );
IF Sta_xrunning AND CT_Rtinput.Q THEN
	 GetSystemTime(udiTimeMs=> CT_Stop, uliTimeUs=> , uliTimeNs=> );
	 IF CT_Start<>0 THEN
	 CT_TEMP := CT_Stop-CT_Start;
	 END_IF
	 CT_Start:=CT_Stop;
END_IF
IF NOT Sta_xrunning THEN
	CT_Stop :=0;
  CT_Start:=0;
	CT_TEMP :=0;
END_IF
CT_TIME:= (UDINT_TO_REAL(CT_TEMP)/1000.0)/CT_number;
END_ACTION

ACTION ACT_status:
IF Sta_safety THEN
   IF Sta_xtart_b THEN
	  Sta_xrunning:=TRUE;
   END_IF
END_IF
END_ACTION

END_FUNCTION_BLOCK

// Device/Application/FC_check/CheckBounds
// 隐含生成代码：不要编辑
FUNCTION CheckBounds : DINT
VAR_INPUT
	index, lower, upper: DINT;
END_VAR

// 隐含生成代码：这里只是对代码实现的建议
IF  index < lower THEN
	CheckBounds := lower;
ELSIF  index > upper THEN
	CheckBounds := upper;
ELSE  
	CheckBounds := index;
END_IF

(*还可以设置断点，日志消息或停止异常情况。
Add CmpApp.library, SysExcept.library and SysTypes2_Itf as newest.
Declaration:
VAR
    _pApp : POINTER TO CmpApp.APPLICATION;
    _result   : SysTypes.RTS_IEC_RESULT;
END_VAR

Implementation:
_pApp := AppGetCurrent(pResult:=_result);
IF  index < lower THEN
        CheckBounds := lower;
        IF _pApp <> 0 THEN
                AppGenerateException(pApp:=_pApp, ulException:=RtsExceptions.RTSEXCPT_ARRAYBOUNDS);
        END_IF
ELSIF  index > upper THEN
        CheckBounds := upper;
        IF _pApp <> 0 THEN
                AppGenerateException(pApp:=_pApp,   ulException:=RtsExceptions.RTSEXCPT_ARRAYBOUNDS);
        END_IF
ELSE  
        CheckBounds := index;
END_IF
*)

END_FUNCTION

// Device/Application/FC_check/CheckDivDInt
// 隐含生成代码：不要编辑
FUNCTION CheckDivDInt : DINT
VAR_INPUT
	divisor:DINT;
END_VAR

// 隐含生成代码：这里只是对代码实现的建议
IF divisor = 0 THEN
	CheckDivDInt:=1;
ELSE
	CheckDivDInt:=divisor;
END_IF;

END_FUNCTION

// Device/Application/FC_check/CheckDivLInt
// 隐含生成代码：不要编辑
FUNCTION CheckDivLInt : LINT
VAR_INPUT
	divisor:LINT;
END_VAR

// 隐含生成代码：这里只是对代码实现的建议
IF divisor = 0 THEN
	CheckDivLInt:=1;
ELSE
	CheckDivLInt:=divisor;
END_IF;

END_FUNCTION

// Device/Application/FC_check/CheckDivReal
// 隐含生成代码：不要编辑
FUNCTION CheckDivReal : REAL
VAR_INPUT
	divisor:REAL;
END_VAR

// 隐含生成代码：这里只是对代码实现的建议
IF divisor = 0 THEN
	CheckDivReal:=1;
ELSE
	CheckDivReal:=divisor;
END_IF;

END_FUNCTION

// Device/Application/FC_check/CheckDivLReal
// 隐含生成代码：不要编辑
FUNCTION CheckDivLReal : LREAL
VAR_INPUT
	divisor:LREAL;
END_VAR

// 隐含生成代码：这里只是对代码实现的建议
IF divisor = 0 THEN
	CheckDivLReal:=1;
ELSE
	CheckDivLReal:=divisor;
END_IF;

END_FUNCTION

// Device/Application/FC_check/CheckPointer
// 隐含生成代码：不要编辑
FUNCTION CheckPointer : POINTER TO BYTE
VAR_INPUT 
	ptToTest : POINTER TO BYTE; // 指针的目标地址
	iSize : DINT;		        // 指针指向的类型大小。（例如：POINTER TO ARRAY [0..9] OF INT为20）
	iGran : DINT;		        // 指针访问的粒度，即指针指向的类型中最大的非结构数据类型的大小。（例如：POINTER TO ARRAY [0..9] OF INT为2）
	bWrite: BOOL;		        // 指示读或写权限。TRUE=写权限。
END_VAR

// 没有标准的实现方式。在此处输入代码
CheckPointer := ptToTest;

END_FUNCTION

// Device/Application/FC_check/CheckRangeSigned
// 隐含生成代码：不要编辑
FUNCTION CheckRangeSigned : DINT
VAR_INPUT
	value, lower, upper: DINT;
END_VAR

